			bStarted := TRUE;
			CASE Mode OF
(*------------------ Read parameter ---------------------------------------------------------------*)
				READWRITEPARAMETERMODE_READ	:
					IF NOT fbAdsRead.Busy THEN
						bStarted := FALSE;
						iState := STATE_RUNNING;
					END_IF;
(*------------------ Write parameter ---------------------------------------------------------------*)
				READWRITEPARAMETERMODE_WRITE	:
					IF NOT fbAdsWrite.BUSY THEN
						bStarted := FALSE;
						iState := STATE_RUNNING;
					END_IF;
			END_CASE;
		ELSE
			Done := FALSE;
			ErrorID := MC_ERROR_COMMAND_NOT_ALLOWED;
			Error := TRUE;
		END_IF;

STATE_RUNNING:  (* wait *)
	IF NOT Error THEN
		CASE Mode OF
		(*------------------ Read parameter ---------------------------------------------------------------*)
			READWRITEPARAMETERMODE_READ	:
				IF fbAdsRead.Err THEN
					ValueLreal := 0.0;
					ValueDword := 0;
					ValueBool := FALSE;
					Done := FALSE;
					ErrorID := fbAdsRead.ErrId;
					Error := TRUE;
					fbAdsRead(READ := FALSE);
					iState := STATE_INITIALIZATION;
				ELSE
					Done := TRUE;
					fbAdsRead(READ := FALSE);
			 		iState:=STATE_INITIALIZATION;
				END_IF;
	(*------------------ Write parameter ---------------------------------------------------------------*)
			READWRITEPARAMETERMODE_WRITE	:
				IF fbAdsWrite.Err THEN
					Done := FALSE;
					ErrorID := fbAdsWrite.ErrId;
					Error := TRUE;
					fbAdsWrite(WRITE := FALSE);
					iState := STATE_INITIALIZATION;
				ELSE
					Done := TRUE;
					fbAdsWrite(WRITE := FALSE);
			 		iState:=STATE_INITIALIZATION;
				END_IF;
		END_CASE;
	ELSE
 		iState:=STATE_INITIALIZATION;
	END_IF;

ELSE  (* CASE : Unknown program state *)
	Error := TRUE;
	ErrorID := 16#FFFFFFFF;
	iState:=STATE_INITIALIZATION;
END_CASE;

ADSbusy := fbAdsWrite.BUSY OR fbAdsRead.BUSY;
IF iState=STATE_INITIALIZATION THEN
	(* reset Busy immediately  when sequence ends *)
	Busy := FALSE;
END_IF
END_FUNCTION_BLOCK

(* POU _FBAXIS_REF, ST *)
(*
	AXIS_REF data structure

	The FBAXIS_REF is actually not a function block but a data structure
	It includes the axis I/O variables as well as additional information.
	The reason for not using a STRUCT is that structures cannot hold
	located I/O variables.
	The user is supposed to use the AXIS_REF data type which internally
	redirects the type to this function block definition (alias).
*)
FUNCTION_BLOCK _FBAXIS_REF
VAR_INPUT
	PlcToNc 	AT %Q* 	: 	PLCTONC_AXIS_REF;
END_VAR
VAR_OUTPUT
	NcToPlc 	AT %I* 	:	NCTOPLC_AXIS_REF;
	ADS	 			: 	ST_AdsAddress;
	Status				:	ST_AxisStatus;
END_VAR
{library private}
VAR
	NcCycleCounter: UDINT;
END_VAR
ReadStatus;
END_FUNCTION_BLOCK
ACTION ReadStatus:
(* NC cycle counter will be incremented after NC task updated the NcToPlc data structure *)
NcCycleCounter := SHR(NcToPlc.OpModeDWord, 24);
(* avoid multiple updates during one cycle which would cause additional CPU load *)
IF NcCycleCounter <> Status.NcCycleCounter OR NcCycleCounter=0 THEN
	Status := _F_ReadStatus( NcToPlc := NcToPlc, PlcToNc := PlcToNc );
END_IF
END_ACTION

(* POU _TCMCGLOBAL, ST *)
(*	Global constants and parameters *)
FUNCTION_BLOCK _TCMCGLOBAL
VAR_INPUT
	NCPORT_TCMC 				:	INT 	:= AMSPORT_R0_NC;
	NCPORT_TCMC_COUPLING	:	INT 	:= AMSPORT_R0_NC; (* used with all axis coupling commands - 12.7.2006 KSt *)
	NCNETID_TCMC 				:	T_AmsNetId := '';
	NCPORT_TCMC_CAM 		:	INT 	:= AMSPORT_R0_NC;
	NCNETID_TCMC_CAM		:	T_AmsNetId := '';
END_VAR
VAR_OUTPUT
END_VAR
VAR CONSTANT
	Axis 	: _ST_NCADS_Axis;	(* IDXGRP and IDXOFFS constants of axis parameter/status/functions *)
	Table 	: _ST_NCADS_Table;	(* IDXGRP and IDXOFFS constants of table parameter/status/functions *)

	NCPORT_TCNCCAMMING_TABLEFUNCTION	: 	UINT	:=	500;

	(* timeout *)
	tTargetPosTimeOut			:	TIME	:= T#6s; (* 20050128 KSt - changed from 5 sec to 6 sec to be later than a NC PEH error (5 sec) *)
	tADSTimeOut   				:	TIME	:= T#1s;

	NCTOPLC_FEEDBACK_MAXWAITCYCLES : INT := 10; (* maximum number of PLC cycles to wait for a cyclic feedback in NcToPlc after an ADS command *)
END_VAR
;
END_FUNCTION_BLOCK

(* POU F_AxisCamDataQueued, ST *)
FUNCTION F_AxisCamDataQueued : BOOL
(* 	reference: 	NC -> PLC axis interface (128 bytes)
	check if bit 22 of an axis StateDWord is set:
	New cam data has been queued to a slave axis which is coupled to master via a cam table. 
	The flag comes up when the PLC modifies the camming data.
	Das Flag wird TRUE, wenn neue bzw. veränderte Kurvenscheibendaten von der SPS an 
	eine Slave-Achse gesendet werden.
*)
VAR_INPUT
	StateDWord : DWORD;
END_VAR
VAR
END_VAR
F_AxisCamDataQueued := (StateDWord AND 2#0000_0000_0100_0000_0000_0000_0000_0000) <> 0;
END_FUNCTION

(* POU F_AxisCamScalingPending, ST *)
FUNCTION F_AxisCamScalingPending : BOOL
(* 	reference: 	NC -> PLC axis interface (128 bytes)
	check if bit 23 of an axis StateDWord is set:
	- The flag signals that the scaling and/or offset setting of a cam table has been requested 
	to be performed 	at a certain master position. This request is pending while the function 
	result is TRUE and has been executed after a falling edge of this signal.
	- Das Flag zeigt an das die Skalierung und/oder das Setzen der Offsets einer Kurvenscheibe
	beauftrag wurde aber erst später (ab einer bestimmten Master-Position) durchgeführt wird.
	Mit fallender Flanke des Signals wurde der Auftrag ausgeführt.
*)
VAR_INPUT
	StateDWord : DWORD;
END_VAR
VAR
END_VAR
F_AxisCamScalingPending := (StateDWord AND 2#0000_0000_1000_0000_0000_0000_0000_0000) <> 0;
END_FUNCTION

(* POU F_AxisCamTableQueued, ST *)
FUNCTION F_AxisCamTableQueued : BOOL
(* 	reference: 	NC -> PLC axis interface (128 bytes)
	check if bit 21 of an axis StateDWord is set:
	New cam data has been queued to a slave axis which is coupled to master via a cam table. 
	The flag comes up when the PLC modifies the camming data.
	Das Flag wird TRUE, wenn neue bzw. veränderte Kurvenscheibendaten von der SPS an 
	eine Slave-Achse gesendet werden.
*)
VAR_INPUT
	StateDWord : DWORD;
END_VAR
VAR
END_VAR
F_AxisCamTableQueued := (StateDWord AND 2#0000_0000_0010_0000_0000_0000_0000_0000) <> 0;
END_FUNCTION

(* POU F_AxisExternalLatchValid, ST *)
FUNCTION F_AxisExternalLatchValid : BOOL
(* 	reference: 	NC -> PLC axis interface (128 bytes)
	check if bit 16 of an axis StateDWord is set:
	External latch value or sensing switch has become valid
	Externer Latchwert bzw. Messtaster gültig geworden
*)
VAR_INPUT
	StateDWord : DWORD;
END_VAR
VAR
END_VAR
F_AxisExternalLatchValid := (StateDWord AND 2#0000_0000_0000_0001_0000_0000_0000_0000) <> 0;
END_FUNCTION

(* POU F_AxisGotNewTargetPosition, ST *)
FUNCTION F_AxisGotNewTargetPosition  : BOOL
(* 	reference: 	NC -> PLC axis interface (128 bytes)
	check if bit 17 of an axis StateDWord is set:
	Axis got a new target position or a new velocity
	while the current move command is in execution.
	Die Zielposition oder die Geschwindigkeit der Achse
	wurde geändert, während die Achse eine Bewegung ausführt
*)
VAR_INPUT
	StateDWord : DWORD;
END_VAR
VAR
END_VAR
F_AxisGotNewTargetPosition := (StateDWord AND 2#0000_0000_0000_0010_0000_0000_0000_0000) <> 0;
END_FUNCTION

(* POU F_AxisHasExtSetPointGen, ST *)
FUNCTION F_AxisHasExtSetPointGen : BOOL
(* 	reference: 	NC -> PLC axis interface (128 bytes)
	check if bit 14 of an axis StateDWord is set:
	Axis has an external set point generator (PLC)
	Achse hat einen externen Sollwertgenerator (SPS)
*)
VAR_INPUT
	StateDWord : DWORD;
END_VAR
VAR
END_VAR
F_AxisHasExtSetPointGen := (StateDWord AND 2#0000_0000_0000_0000_0100_0000_0000_0000) <> 0;
END_FUNCTION

(* POU F_AxisInPTPmode, ST *)
FUNCTION F_AxisInPTPmode : BOOL
(* 	reference: 	NC -> PLC axis interface (128 bytes)
	check if bit 25 of an axis StateDWord is set:
	- The flag signals that the axis accepts PTP motion commands. That requires that the axis is 
	not coupled to other axes and not part of a NC-I or FIFO group.
	- Das Flag zeigt an, dass die Achse PTP Bewegungskommandos entgegen nimmt. Das setzt 
	voraus, dass die Achse nicht gekoppelt ist oder in eine NC-I oder FIFO-Gruppe integriert ist.
*)
VAR_INPUT
	StateDWord : DWORD;
END_VAR
VAR
END_VAR
F_AxisInPTPmode := (StateDWord AND 2#0000_0010_0000_0000_0000_0000_0000_0000) <> 0;
END_FUNCTION

(* POU F_AxisIoDataIsInvalid, ST *)
FUNCTION F_AxisIoDataIsInvalid : BOOL
(* 	reference: 	NC -> PLC axis interface (128 bytes)
	check if bit 30 of an axis StateDWord is set:
	Axis I/O data is invalid  (e.g. invalid 'WcState' or 'CdlState' )
	Achse hat keine gültigen I/O-Daten  (e.g. invalid 'WcState' or 'CdlState' )
*)
VAR_INPUT
	StateDWord : DWORD;
END_VAR
VAR
END_VAR
F_AxisIoDataIsInvalid := (StateDWord AND 2#0100_0000_0000_0000_0000_0000_0000_0000) <> 0;
END_FUNCTION

(* POU F_AxisIsCalibrated, ST *)
FUNCTION F_AxisIsCalibrated : BOOL
(* 	reference: 	NC -> PLC axis interface (128 bytes)
	check if bit 1 of an axis StateDWord is set:
	Axis has been referenced ("Axis calibrated")
	Achse ist referenziert ("Achse geeicht")
*)
VAR_INPUT
	StateDWord : DWORD;
END_VAR
VAR
END_VAR
F_AxisIsCalibrated := (StateDWord AND 2#0000_0000_0000_0000_0000_0000_0000_0010) <> 0;
END_FUNCTION

(* POU F_AxisIsMoving, ST *)
FUNCTION F_AxisIsMoving : BOOL
(* 	reference: 	NC -> PLC axis interface (128 bytes)
	check if bit 9 OR 10 of an axis StateDWord is set:
	Axis moving (forward or backwards)
	Achse fährt (vorwärts oder rückwärts)
*)
VAR_INPUT
	StateDWord : DWORD;
END_VAR
VAR
END_VAR
F_AxisIsMoving := (StateDWord AND 2#0000_0000_0000_0000_0000_0110_0000_0000) <> 0;
END_FUNCTION

(* POU F_AxisIsMovingBackwards, ST *)
FUNCTION F_AxisIsMovingBackwards : BOOL
(* 	reference: 	NC -> PLC axis interface (128 bytes)
	check if bit 10 of an axis StateDWord is set:
	Axis moving to logically smaller values
	Achse fährt logisch kleiner
*)
VAR_INPUT
	StateDWord : DWORD;
END_VAR
VAR
END_VAR
F_AxisIsMovingBackwards := (StateDWord AND 2#0000_0000_0000_0000_0000_0100_0000_0000) <> 0;
END_FUNCTION

(* POU F_AxisIsMovingForward, ST *)
FUNCTION F_AxisIsMovingForward : BOOL
(* 	reference: 	NC -> PLC axis interface (128 bytes)
	check if bit 9 of an axis StateDWord is set:
	Axis moving to logically larger values
	Achse fährt logisch größer
*)
VAR_INPUT
	StateDWord : DWORD;
END_VAR
VAR
END_VAR
F_AxisIsMovingForward := (StateDWord AND 2#0000_0000_0000_0000_0000_0010_0000_0000) <> 0;
END_FUNCTION

(* POU F_AxisIsNotMoving, ST *)
FUNCTION F_AxisIsNotMoving : BOOL
(* 	reference: 	NC -> PLC axis interface (128 bytes)
	check if bit 2 of an axis StateDWord is set:
	Axis is logically stationary ("Axis not moving")
	Achse ist im logischen Stillstand ("Achse fährt nicht")
*)
VAR_INPUT
	StateDWord : DWORD;
END_VAR
VAR
END_VAR
F_AxisIsNotMoving := (StateDWord AND 2#0000_0000_0000_0000_0000_0000_0000_0100) <> 0;
END_FUNCTION

(* POU F_AxisJobPending, ST *)
FUNCTION F_AxisJobPending : BOOL
(* 	reference: 	NC -> PLC axis interface (128 bytes)
	check if bit 24 of an axis StateDWord is set:
	- The flag signals that the a new motion job ist pending and will be 
	   executed after the active job is finished (buffer mode)
	- Das Flag zeigt an das die ein neuer Fahrauftrag gepuffert ist,
	   um nach dem aktuellen Auftrag ausgeführt zu werden (buffer mode)
*)
VAR_INPUT
	StateDWord : DWORD;
END_VAR
VAR
END_VAR
F_AxisJobPending := (StateDWord AND 2#0000_0001_0000_0000_0000_0000_0000_0000) <> 0;
END_FUNCTION

(* POU F_AxisReachedConstantVelocity, ST *)
FUNCTION F_AxisReachedConstantVelocity  : BOOL
(* 	reference: 	NC -> PLC axis interface (128 bytes)
	check if bit 12 of an axis StateDWord is set:
	Axis has reached its constant velocity or rotary speed
	Achse hat V-Konst bzw. Drehzahl erreicht
*)
VAR_INPUT
	StateDWord : DWORD;
END_VAR
VAR
END_VAR
F_AxisReachedConstantVelocity := (StateDWord AND 2#0000_0000_0000_0000_0001_0000_0000_0000) <> 0;
END_FUNCTION

(* POU F_GetVersion_TcMC2, ST *)
FUNCTION F_GetVersion_TcMC2 : UINT	(* Gets the library version info *)
VAR_INPUT
	nVersionElement		:	INT;
END_VAR
(*
	Possible nVersionElement parameter:
	1	:	major number
	2	:	minor number
	3	:	revision number
*)

(* Version history:
Date	|	Version/Author |	Remark
----------------------------------------------------------------------------------------------------
11.09.01	|	2.01 JP		|	new version depending on 0.99D
22.11.01	|	2.02 JP		|	new version depending on 0.99F
18.01.02	|	2.03 JP		|	new version depending on 1.0
		|				|	changed names, interfaces, execute behavior
25.01.02	|	2.04 JP		|	no CAMMING, change behavior of MC_Power
07.02.02	|	2.05 JP		|	SetOverride in unit less than 1%
13.02.02	|	2.06 JP		|	New: MC_NewPos and MC_NewPosAndVelo
		|				|	removed MC_MoveAdditive
14.02.02	|	2.07 JP		|	completed: MC_Home, MC_MoveSuperImposed
14.02.02	|	2.08 JP		|	renamed MC_NewPosAndVelo New: MC_SetOverride edge triggered
15.02.02	|	2.09 JP		|	changed: MC_Gear
15.02.02	|	2.10 JP		|	changed: MC_SetOverride
04.04.02	|	2.11 JP		|	changed: done for MC_Home 
		|				|	new: Check TimeOut for MoveAbsolute, MoveRelative, Home
08.03.02	|	2.12 JP		|	changed: new flag inserted 
12.03.02	|	2.13 JP		|	changed: reset of bNotExecute
18.03.02	|	2.14 JP		|	changed: MC_Reset waits for ready
22.03.02	|	2.15 JP		|	changed: MC_Read and Write FBs
26.03.02	|	2.16 JP		|	revised: Read/Write Parameter FBs
27.03.02	|	2.17 JP		|	revised: Read/Write Parameter FBs and Home (calibration cam)
09.04.02	|	2.18 JP		|	changed parameter type of some parameters
17.04.02	|	2.19 JP		|	changed: Read(Bool)Parameter new Input to select read mode
							Boolean parameters can be read with ReadParameter
							changed MC_Power: new input override !!			
23.04.02	|	2.20 JP		|	fixed: MC_Home changed: Behavior of MC_MoveAbsolute/Relative
25.04.02	|	2.21 JP		|	changed: MC_Reset: now not waiting for 'axis is ready'. Check with MC_Power !
26.04.02	|	2.22 JP		|	MC_Home: If Posistion =  DEFAULT_HOME_POSITION --> no set of position
							MC_MoveXX: more detailed error messages
05.07.02	|	2.23 JP		|	new MC_MoveAbsoluteOrRestart: combines MoveAbsolute and NewPos
19.07.02	|	2.24 JP		|	changed: E_STATES ---> E_TCMC_STATES
12.09.02	|	2.25 KST		|	changed: MC_MoveAbsolute and MC_MoveRelative now based on FB_MoveGeneric
							MC_NewPos and MC_NewPosAndVelo based on new FB_NewPosAndVeloGeneric 
							new internal start types in MC_MoveAbsoluteOrRestart (message suppression)
16.09.02	|	2.26 ChristophC|	changed: MC_SetActualPosition due to changes in TcNC.Lib
16.10.02	|	2.27 KST		|	new: MC_ExtSetPointGenEnable and MC_ExtSetPointGenDisable
29.10.02	|	2.28 ChristophC|	MC_Stop and MC_SetActualPosition: Ads port changed from TcMcGlobal.NCPORT_TCMC => AMSPORT_R0_NCSAF
12.11.02	|	2.29 ChristophC|	MC_OverrideFilter function block added
13.12.02	|	2.30 JP		|	several smaller changes: MC_ReadStatus, MC_Stop
22.01.03	|	2.31 KSt		|	new additional function MC_ExtSetPointGenFeed
24.03.03	|	2.32 JP		|	added: MC_GearFloat, corr. MC_ReadBoolParameter (wrong for AxisEnPostionRangeMonitoring)
26.03.03	|	2.33 KSt		|	added: MC_MoveModulo
04.04.03	|	2.34 KSt		|	changed: MC_MoveAbsoluteOrRestart, Done will be reset at once after Execute=FALSE
12.05.03	|	2.35 JP		|	changed: MC_MoveVelocity, MC_Home (error handling), MC_ReadStatus
14.05.03	|	2.36 KSt		|	changed: MC_Home, MC_MoveAbsoluteOrRestart
15.05.03	|	2.36.1 KSt	|	changed: MC_Home
28.05.03	|	2.37 KSt		|	changed: MC_MoveVelocity, abort during acceleration phase	
							changed: MC_MoveAbsoluteOrRestart, reset internal error on restart
27.06.03	|	2.38 JP		|	changed: MC_Stop: Execute behavior
22.07.03	|	2.38.1 KSt	|	added: new error codes
12.08.03	|	2.39 KSt		|	changed: FB_ReadWriteParameter, size of bool parameters
15.08.03	|	2.40 KSt		|	added: new block MC_ChangeDynParam
19.08.03	|	2.41 JP		|	changed: MC_ReadParameter: Done falls with Execute
01.10.03	|	2.42 KSt		|	changed: MC_MoveAbsoluteOrRestart, Execute directly after done issue fixed
09.10.03	|	2.43 KSt		|	new function block MC_SetReferenceFlag
04.12.03	|	2.44 KSt		|	ReadBoolParameter(AxisEnTargetPositionMonitoring) corrected
12.01.04	|	2.45 KSt		|	MC_MoveSuperimposed revised
						|	R_Trigger(execute) moved outside CASE in all move function blocks
19.01.04	|	2.45.1 KSt	|	Busy Signal in MC_MoveSuperimposed
30.04.04	|	2.46.0 KSt	|	New function blocks MC_TouchProbe, MC_AbortTrigger, internal block MC_OrientedStop
						|	MC_ReadParameter revised
06.05.04	|	2.46.1 KSt	|	Correction in MC_OrientedStop
21.05.04	|	2.47.0 KSt	|	MC_GearInDyn added - master slave coupling with dynamic gear ratio
06.08.04	|	2.47.1 KSt	|	MC_OrientedStop moved from internal to additional folder
						|	MC_MoveAbsoluteOrRestart additional internal error code NC_ERROR_STARTINTERNAL_NOTREADY evaluated
23.08.04	|	2.47.2 KSt	|	new local flag EmergencyStop in MC_Stop signals type of internal ADS stop command
10.01.05	|	2.47.3 KSt	|	new function block MC_MoveSuperImposedExt
28.01.05	|	2.47.4 KSt	|	TcMcGlobal.tTargetPosTimeOut changed from 5 sec to 6 sec to be later than a NC PEH error (5 sec)
15.02.05	|	2.48.0 KSt	|	new function block MC_GearOutExt 
28.02.05	|	2.49.0 JP		|	Execute and Done behavior corrected for MC_ReadActualPos and MC_SetActualPos
10.03.05	|	2.50.0 KSt	|	all function blocks use a global AMS net-ID TcMcGlobal.NCNETID_TCMC which may be modified by the user
17.03.05	|	2.51.0 KSt	|	new function block MC_PowerStepper
						|	MC_MoveAbsoluteOrRestart restart while starting (adswrite.Busy) changed
24.05.05	|	2.52.0 KSt	|	acceleration added to block MC_GearOutExt 
05.07.05	|	2.53.0 KSt	|	new local flag ADSbusy in all function blocks
05.07.05	|	2.54.0 KSt	|	new function block MC_GearInDynCCV
06.07.05	|	2.55.0 KSt	|	Busy timing improved in all function blocks (turns immediately to FALSE with Done or Error or Aborted)
25.07.05	|	2.55.1 KSt	|	Change for status output behavior 
26.07.05	|	2.55.2 KSt	|	MC_GearOutExt extended through mode 'oriented stop'
03.08.05	|	2.55.3 KSt	|	Commands MC_MoveAbsoluteOrRestart, MC_NewPos and MC_NewPosAndVelo now directed to port AMSPORT_R0_NCSAF
						|	Summary of other commands to SAF: MC_Stop, MC_OrientedStop, MC_TouchProbe, MC_AbortTrigger, MC_SetReferenceFlag, MC_PowerStepper
14.09.05	|	2.56.0 KSt	|	new function block MC_ParameterizedStop
26.09.05	|	2.56.1 KSt	|	Jerk parameter added to MC_ChangeDynParam. Block moved into the internal folder.
07.11.05	|	2.56.2 KSt	|	internal block FB_ReadCharacteristicValues changed to ADSRDWRT
19.12.05	|	2.56.3 KSt	|	new block MC_SetActualPositionOnTheFly
05.01.06	|	2.56.4 KSt	|	new blocks MC_ReadParameterSet and MC_ReadAxisComponents
21.02.06	|	2.57.0 KSt	|	NC status feedback monitoring changed in MC_GearIn and MC_GearInFloat
29.03.06	|	2.57.1 KSt	|	new order of the blocks in the library tree
11.04.06	|	2.57.2 HKP	|	Command MC_ChangeDynParam now directed to port AMSPORT_R0_NCSAF
10.05.06	|	2.57.3 KSt	|	new function block MC_Jog
17.05.06	|	2.57.4 KSt	|	MC_Jog: MC_JOGMODE_INCHING_MODULO temporarily deactivated
05.07.06	|	2.57.5 KSt	|	NC status feedback monitoring changed in MC_GearInDyn and MC_GearInDynCCV
=======	|===============	|==========================================================================
12.07.06	|	2.57.6 KSt	|	new AMS port NCPORT_TCMC_COUPLING for all coupling commands
11.08.06	|	2.57.7 KSt	|	reset Done when Execute is FALSE in FB_NewPosAndVeloGeneric
						|	MC_Jog released
22.08.06	|	2.57.8 KSt	|	new function block MC_AbortSuperposition
07.11.06	|	2.57.9 HKP	|	changes in function block MC_PowerStepper
06.02.07	|	2.57.10 KSt	|	initialization problem with modulo positions fixed in MC_TouchProbe.
						|	recorded position at PlcEvent now modulo when requested.
14.03.07	|	2.57.11 KSt	|	MC_Jog: Handling of CommandAborted corrected
24.04.07	|	2.57.12 KSt	|	additional parameters in MC_AxisPara, MC_ReadParameters, MC_WriteParameters
31.05.07	|	2.57.13 KSt	|	FPU exception with LREAL_TO_BOOL and DWORD_TO_BOOL fixed in FB_ReadWriteParameter 
12.06.07	|	2.57.14 KSt	|	FB_NewPosAndVeloGeneric and MC_MoveSuperImposed(Ext): IF condition changed from "NOT AxisIsMoving" to "NOT AxisHasJob"
=======	|===============	|==========================================================================
12.06.07	|	2.57.14 KSt	|	TcMC2 development started - following 2.xx.xx changes have been added in parallel
02.11.07	|	2.57.15 KSt	|	data structure ST_TableCharacValues extended
18.12.07	|	2.57.16 KSt	|	MC_Jog is now internally using MC_MoveRelative instead of MC_MoveAbsolute to work with backlash compensation
20.05.08	|	2.57.18 KSt	|	AxisModuloPositionFlag added to MC_ReadBoolParameter
17.06.08	|	2.57.20 KSt	|	MC_GearInMultiMaster added
24.07.08	|	2.57.22 KSt	|	MC_Power supports now a minimum Enable-Off/On toggle time of 50ms to reenable the Status output
28.10.08	|	2.57.23 KSt	|	new function block MC_SetEncoderScalingFactor
=======	|===============	|==========================================================================
16.03.07	|	3.00.00 KSt	|	new version depending on PLCopen V1.1 (beta)
25.08.08   |	3.00.01 KSt	|	released as TcMC2 
17.09.08   |	3.00.02 KSt	|	last result added in MC_Reset
26.11.08   |	3.00.03 KSt	|	change in MC_Stop and MoveGeneric for delayed error handling
01.12.08   |	3.00.04 KSt	|	MC_Stop - Done is set immediately at standstill
18.12.08   |	3.00.05 KSt	|	MC_Power - uses now ControlLoopClosed instead of AxisIsReady
13.01.09   |	3.00.06 KSt	|	independent characteristic data for camming and flying saw
16.01.09   |	3.00.07 KSt	|	all move commands: changed handling of CmdNo=0 and CmdNo+2 leads to better results (CommandAborted)
23.01.09   |	3.00.08 KSt	|	MC_MoveSuperimposed is now passed to port AMSPORT_R0_NCSAF (501)
28.01.09   |	3.00.09 KSt	|	Homing mode MC_Direct added - Mode option for MC_SetPosition added
29.01.09   |	3.00.10 KSt	|	Warning output added to MC_MoveSuperimposed
05.02.09   |	3.00.11 KSt	|	axis state is now DISABLED if control loop is not closed (was STANDSTILL for virtual axes - _F_AxisState)
05.02.09   |	3.00.11 KSt	|	all move commands: CmdNo=0 is ignored as invalid - change of the coupled state leads to CommandAborted
06.02.09   |	3.00.11 KSt	|	errors on missing cyclic NC command feedback are delayed for a few cycles to avoid problems with multiple function block calls during one PLC cycle
19.02.09   |	3.00.12 KSt	|	MC_GearInDyn and MC_GearInMultimaster - no reset of gear ratio after Enable is reset to FALSE
24.02.09   |	3.01.00 KSt	|	Motion commands on slaves (must be enabled in the axis parameters before)
12.03.09   |	3.01.01 KSt	|	MC_Jog - Active output added - reset outputs when Execute is false 
09.04.09   |	3.01.02 KSt	|	MC_SetPosition and MC_SetEncoderScalingFactor - explicit encoder / control loop index 0..n can be selected
15.04.09   |	3.01.03 KSt	|	MC_Stop - outputs (except Busy) are reset after Execute=FALSE - can be retriggered during release phase
17.04.09   |	3.01.04 KSt	|	MC_Home - static homing with DEFAULT_HOME_POSITION implemented - Option.ClearPositionLag available 
11.05.09   |	3.01.05 KSt	|	MC_Stop - incorrect error message 4B63 removed;  
30.06.09   |	3.01.06 KSt	|	MC_MoveSuperimposed - new types ACCREDUCTION - new AbortOptions
28.07.09   |	3.01.07 KSt	|	MC_ExtSetPointGenFeed feeds additional counter information to the NC
13.08.09   |	3.01.08 KSt	|	MC_MoveSuperimposed - new AbortOptions - Done behavior adapted
01.09.09   |	3.01.09 KSt	|	MC_SetPosition - new option 'set absolute measuring'
30.09.09   |	3.01.10 KSt	|	MC_MoveSuperimposed - fix for new AbortOptions - HasJob flag not required before starting the command
06.10.09   |	3.01.11 KSt	|	MC_Stop - wait extra cycles before axis release error 
06.10.09   |	3.01.12 KSt	|	MC_MoveSuperimposed - fix for new AbortOptions - HasJob or IsMoving check at beginning and end of compensation 
07.10.09   |	3.01.13 KSt	|	MC_MoveSuperimposed - initial motion check removed for new AbortOptions
28.10.09   |	3.01.14 KSt	|	MC_ExtSetPointGenEnable/Disable - port changed from SVB to SAF
06.11.09   |	3.01.15 KSt	|	MC_SetPosition - new option 'set absolute measuring' removed
09.11.09   |	3.01.16 KSt	|	MC_Stop on slave axes was not rejected with error - fixed
18.11.09   |	3.01.17 KSt	|	MC_Jog - usage with protected (coupled) axes refused
26.11.09   |	3.01.18 KSt	|	Axis status data: UpdateCycleTime calculation fixed
08.12.09   |	3.01.19 KSt	|	_FB_MoveGeneric - mapping check to avoid early Error and CommandAborted signals
25.02.10   |	3.01.20 KSt	|	MC_MoveSuperimposed - additional outputs ActualAcceleration and ActualDeceleration
11.03.10   |	3.01.21 KSt	|	MC_Power - no Enable timeout error for coupled axes
*)
CASE nVersionElement OF
1:	(* major number *)
	F_GetVersion_TcMC2 := 3;
2:	(* minor number *)
	F_GetVersion_TcMC2 := 1;
3:	(* revision number *)
	F_GetVersion_TcMC2 := 21;
ELSE
	F_GetVersion_TcMC2 := 16#FFFF;
END_CASE
END_FUNCTION

(* POU MC_AbortSuperposition, ST *)
FUNCTION_BLOCK MC_AbortSuperposition
VAR_INPUT
	Execute		:	BOOL;	(* Starts touch probe recording *)
END_VAR
VAR_OUTPUT
	Done		:	BOOL;	(* move completed *)
	Busy		: 	BOOL;	(* function block is currently Busy *)
	Error		:	BOOL;	(* Signals that error has occured within Function Block *)
	ErrorID		:	UDINT;	(* Error identification *)
END_VAR
VAR_IN_OUT
	Axis			:	AXIS_REF; (* Identifies the axis of which the position should be recorded at a defined event at the trigger input *)
END_VAR
VAR
	LastExecutionResult: 	_ST_FunctionBlockResults;
	ADSbusy	: 	BOOL;
	fbOnTrigger	: 	R_TRIG;
	fbADSwrite	: 	ADSWRITE;
	iState		:	_E_TcMC_STATES := STATE_INITIALIZATION;
END_VAR
fbOnTrigger(CLK:= Execute);

CASE iState OF
STATE_INITIALIZATION: (* initial iState *)
	Busy := FALSE;
	IF NOT Execute THEN
		Done := FALSE;
		Error := FALSE;
		ErrorID := 0;
	END_IF
	IF fbOnTrigger.Q THEN
		Busy := TRUE;
		(* initialization *)
		Done := FALSE;
		Error := FALSE;
		ErrorID := 0;
		LastExecutionResult.Done := FALSE;
		LastExecutionResult.CommandAborted := FALSE;
		LastExecutionResult.Error := FALSE;
		LastExecutionResult.ErrorID := 0;
		fbADSwrite(WRITE:=FALSE);
		fbADSwrite(	NETID:= TcMcGlobal.NCNETID_TCMC,
					PORT:=TcMcGlobal.NCPORT_TCMC ,
					IDXGRP:= TcMcGlobal.Axis.Functions.IDXGRP + Axis.NcToPlc.AxisId,
					IDXOFFS:= TcMcGlobal.Axis.Functions.IDXOFFS.STOPSCOM,	(* abort superposition *)
					LEN:=0,
					SRCADDR:=0,
					WRITE:=TRUE ,
					TMOUT:= TcMcGlobal.tADSTimeOut);
		iState := STATE_ORDER;
	END_IF

STATE_ORDER:  (* wait until command is accepted *)
	fbADSwrite(WRITE:= TRUE);
	IF NOT fbADSwrite.BUSY THEN
		Error := fbADSwrite.ERR;
		ErrorID := fbADSwrite.ERRID;
		IF NOT Error THEN
			IF NOT F_AxisIsCompensating(Axis.NcToPlc.StateDWord) THEN
				Done := TRUE;
				Busy := FALSE;
				iState := STATE_INITIALIZATION;
			ELSE
				iState := STATE_RUNNING;
			END_IF
		ELSE
			Busy := FALSE;
			iState := STATE_INITIALIZATION;
		END_IF
		LastExecutionResult.Done := Done;
		LastExecutionResult.Error := Error;
		LastExecutionResult.ErrorID := ErrorID;
	END_IF

STATE_RUNNING:
	IF NOT F_AxisIsCompensating(Axis.NcToPlc.StateDWord) THEN
		Done := TRUE;
		Busy := FALSE;
		LastExecutionResult.Done := Done;
		LastExecutionResult.Error := Error;
		LastExecutionResult.ErrorID := ErrorID;
		iState := STATE_INITIALIZATION;
	END_IF
END_CASE

ADSbusy := fbAdsWrite.BUSY;
END_FUNCTION_BLOCK

(* POU MC_AbortTrigger, ST *)
FUNCTION_BLOCK MC_AbortTrigger
(*	The function block is used to abort function blocks which are connected to
	trigger events (e.g. MC_TouchProbe) 
*)
VAR_IN_OUT
	Axis			:	AXIS_REF; 		(* B *)	(* Identifies the axis of which the position should be recorded at a defined event at the trigger input *)
	TriggerInput	: 	TRIGGER_REF; 	(* E *)	(* Reference to the trigger signal source. *)
END_VAR
VAR_INPUT
	Execute		:	BOOL;	(* B *)	(* Starts aborting  touch probe sequence *)
END_VAR
VAR_OUTPUT
	Done		:	BOOL;	(* B *)	(* function completed *)
	Busy		: 	BOOL;	(* E *)	(* function block is currently Busy *)
	Error		:	BOOL;	(* B *)	(* Signals that error has occurred within Function Block *)
	ErrorID		:	UDINT;	(* E *)	(* Error identification *)
END_VAR
VAR
	ADSbusy	: 	BOOL;
	fbADSwrite	: 	ADSWRITE;
END_VAR
{library private}
VAR CONSTANT
	OLDADSINTERFACE : BOOL := TRUE; (* temporary flag to test old and new NC ADS touch probe interface *)
END_VAR
VAR
	LatchID		: 	UDINT;
	fbOnTrigger	: 	R_TRIG;
END_VAR
IF NOT Execute THEN
	Done := FALSE;
	Error := FALSE;			(* reset at falling edge of Execute *)
	ErrorID := 0;
END_IF

fbOnTrigger(CLK:= Execute);
IF fbOnTrigger.Q OR fbADSwrite.BUSY THEN
	Busy := TRUE;
	IF fbOnTrigger.Q THEN
		(* initialization *)
		Done := FALSE;
		Error := FALSE;
		ErrorID := 0;
		fbADSwrite(WRITE:=FALSE);
		IF TriggerInput.EncoderID > 255 THEN
			Error := TRUE;
			ErrorID := MC_ERROR_INVALID_TOUCH_PROBE;
		END_IF
	END_IF

	IF NOT Error THEN
		CASE TriggerInput.TouchProbe OF
			TouchProbe1,
			TouchProbe2,
			TouchProbe3,
			TouchProbe4:
			LatchID := TriggerInput.TouchProbe;
			fbADSwrite(	NETID:= TcMcGlobal.NCNETID_TCMC,
						PORT:=AMSPORT_R0_NCSAF ,
						IDXGRP:=16#5200+TriggerInput.EncoderID ,
						IDXOFFS:=16#205,	(* deactivate touch probe *)
						LEN:=SEL(OLDADSINTERFACE, SIZEOF(LatchID), 0) ,
						SRCADDR:=ADR(LatchID),
						WRITE:=TRUE ,
						TMOUT:=TcMcGlobal.tADSTimeOut);
			IF NOT fbADSwrite.BUSY THEN
				Error := fbADSwrite.ERR;
				ErrorID := fbADSwrite.ERRID;
				TriggerInput.ProbeState := SEL(Error, TouchProbeAborted, TriggerInput.ProbeState );
				Done := NOT Error;
			END_IF

			PlcEvent:
				(* no action necessary here *);
				TriggerInput.ProbeState := TouchProbeAborted;
				Done := TRUE;

			ELSE (* case *)
				Error := TRUE;
				ErrorID := MC_ERROR_INVALID_TOUCH_PROBE;
		END_CASE
	END_IF
ELSE
	Busy := FALSE;
END_IF

ADSbusy := fbAdsWrite.BUSY;
(* reset Busy immediately  when sequence ends *)
Busy := fbOnTrigger.Q OR fbADSwrite.BUSY;
END_FUNCTION_BLOCK

(* POU MC_ExtSetPointGenDisable, FBD *)
FUNCTION_BLOCK MC_ExtSetPointGenDisable
VAR_IN_OUT
	Axis	:	AXIS_REF;
END_VAR
VAR_INPUT
	Execute : BOOL;
END_VAR
VAR_OUTPUT
	Done : BOOL;
	Busy: BOOL;
	Error: BOOL;
	ErrorID: UDINT;
	Enabled: BOOL;
END_VAR
VAR
	ADSbusy: BOOL;
	Disable: ADSWRITE;
	RunOnce: BOOL;
END_VAR
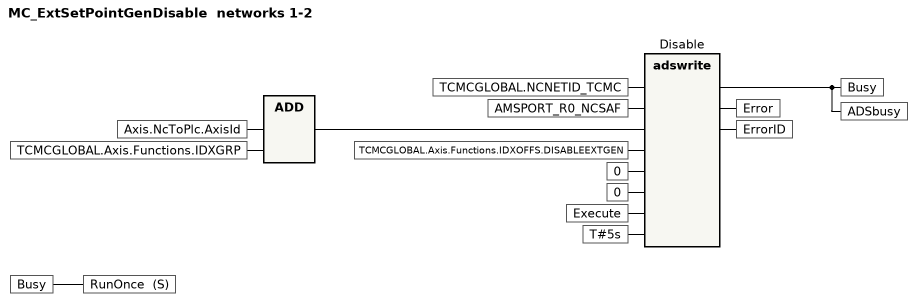
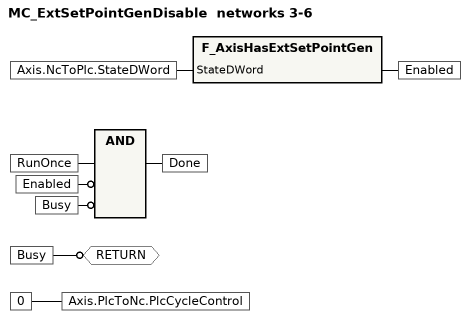
_FBD_ (* Function Block Diagram *)
NETWORK 1 (* ( * 2009-10-28 KSt - port changed from SVB to SAF * ) *)
	Disable:adswrite(TCMCGLOBAL.NCNETID_TCMC, AMSPORT_R0_NCSAF, ADD(Axis.NcToPlc.AxisId, TCMCGLOBAL.Axis.Functions.IDXGRP), TCMCGLOBAL.Axis.Functions.IDXOFFS.DISABLEEXTGEN, 0, 0, Execute, T#5s, out 2 => Error, out 3 => ErrorID) => Busy, ADSbusy
NETWORK 2
	Busy => S RunOnce
NETWORK 3
	F_AxisHasExtSetPointGen(StateDWord: Axis.NcToPlc.StateDWord) => Enabled
NETWORK 4
	AND(RunOnce, NOT Enabled, NOT Busy) => Done
NETWORK 5
	NOT Busy => <RETURN>
NETWORK 6
	0 => Axis.PlcToNc.PlcCycleControl
_END_FBD_
END_FUNCTION_BLOCK

(* POU MC_ExtSetPointGenEnable, FBD *)
FUNCTION_BLOCK MC_ExtSetPointGenEnable
VAR_IN_OUT
	Axis	:	AXIS_REF;
END_VAR
VAR_INPUT
	Execute : BOOL;
	Position : LREAL;
	PositionType : E_PositionType;
END_VAR
VAR_OUTPUT
	Done : BOOL;
	Busy: BOOL;
	Error: BOOL;
	ErrorID: UDINT;
	Enabled: BOOL;
END_VAR
VAR
	ADSbusy: BOOL;
	Enable: ADSWRITE;
	sExtSetPointGen : _ST_TcNC_SetPos;
END_VAR
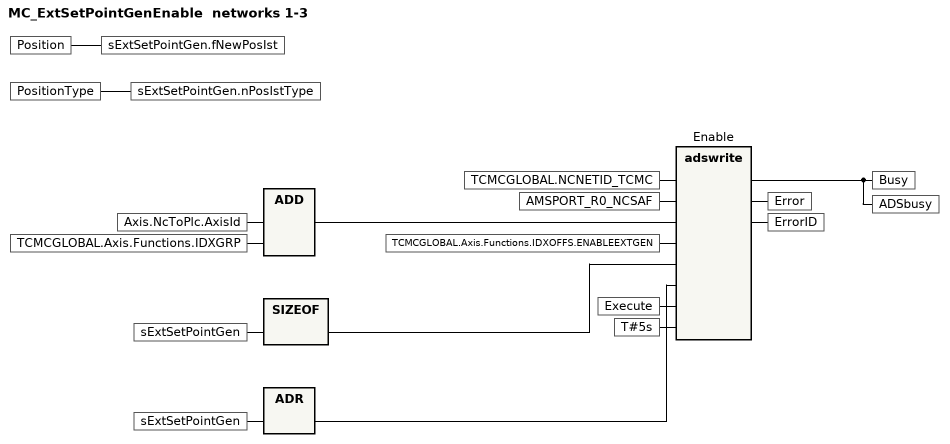
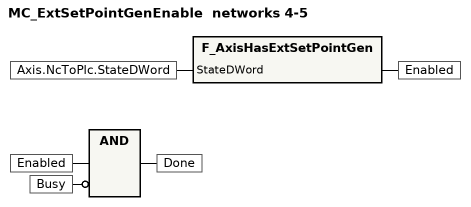
_FBD_ (* Function Block Diagram *)
NETWORK 1
	Position => sExtSetPointGen.fNewPosIst
NETWORK 2
	PositionType => sExtSetPointGen.nPosIstType
NETWORK 3 (* ( * 2009-10-28 KSt - port changed from SVB to SAF * ) *)
	Enable:adswrite(TCMCGLOBAL.NCNETID_TCMC, AMSPORT_R0_NCSAF, ADD(Axis.NcToPlc.AxisId, TCMCGLOBAL.Axis.Functions.IDXGRP), TCMCGLOBAL.Axis.Functions.IDXOFFS.ENABLEEXTGEN, SIZEOF(sExtSetPointGen), ADR(sExtSetPointGen), Execute, T#5s, out 2 => Error, out 3 => ErrorID) => Busy, ADSbusy
NETWORK 4
	F_AxisHasExtSetPointGen(StateDWord: Axis.NcToPlc.StateDWord) => Enabled
NETWORK 5
	AND(Enabled, NOT Busy) => Done
_END_FBD_
(* the same logic as Structured Text *)
(* Network 1 *)
sExtSetPointGen.fNewPosIst := Position;
(* Network 2 *)
sExtSetPointGen.nPosIstType := PositionType;
(* Network 3: see the listing above *)
(* Network 4 *)
Enabled := F_AxisHasExtSetPointGen(StateDWord := Axis.NcToPlc.StateDWord);
(* Network 5 *)
Done := Enabled AND NOT Busy;
END_FUNCTION_BLOCK

(* POU MC_ExtSetPointGenFeed, ST *)
FUNCTION MC_ExtSetPointGenFeed : BOOL
VAR_IN_OUT
	Axis	:	AXIS_REF;
END_VAR
VAR_INPUT
	Position		: LREAL;
	Velocity		: LREAL;
	Acceleration	: LREAL;
	Direction 	: DINT;
END_VAR
VAR
	GetTaskIndex : GETCURTASKINDEX;
END_VAR
Axis.PlcToNc.ExtSetPos := Position;
Axis.PlcToNc.ExtSetVelo := Velocity;
Axis.PlcToNc.ExtSetAcc := Acceleration;
Axis.PlcToNc.ExtSetDirection := Direction;

GetTaskIndex();
Axis.PlcToNc.PlcCycleControl.0 := 1; (* activate PLC cycle information to NC *)
Axis.PlcToNc.PlcCycleControl.1 := SystemTaskInfoArr[ GetTaskIndex.index ].cycleTimeExceeded;
Axis.PlcToNc.PlcCycleCount := Axis.PlcToNc.PlcCycleCount + 1;
END_FUNCTION

(* POU MC_GearIn, ST *)
FUNCTION_BLOCK MC_GearIn
(*	This Function Block commands a ratio between the velocity of the slave and master axis. *)
VAR_IN_OUT
	Master			:	AXIS_REF;	(* B *)
	Slave			:	AXIS_REF;	(* B *)
END_VAR
VAR_INPUT
	Execute			:	BOOL;	(* B *)
	RatioNumerator	:	LREAL	(* B *)	:= 1; (* changed from INT (PLCopen) to LREAL *)
	RatioDenominator	:	UINT	(* B *)	:= 1;
	Acceleration		:	LREAL;	(* E *)
	Deceleration		:	LREAL;	(* E *)
	Jerk				:	LREAL;	(* E *)
	BufferMode		:	MC_BufferMode;	(* E *)
	Options			: 	ST_GearInOptions;	(* V *)	(* optional parameters *)
END_VAR
VAR_OUTPUT
	InGear			:	BOOL;	(* B *)
	Busy			: 	BOOL;	(* E *)
	Active			: 	BOOL;	(* E *)
	CommandAborted	:	BOOL;	(* E *)
	Error			:	BOOL;	(* B *)
	ErrorID			:	UDINT;	(* E *)
END_VAR
VAR
	LastExecutionResult	: 	_ST_FunctionBlockResults;
	ADSbusy: BOOL;
	iState				:	_E_TcMC_STATES := STATE_INITIALIZATION;
	fbAdsWrite			:	ADSWRITE;
	sCouple				:	_ST_TcNC_CoupleSlave;
	fbOptGearInDyn		: 	MC_GearInDyn;
END_VAR
{library private}
VAR
	fbOnTrigger			:	R_TRIG;
	TimerStateFeedback	: 	TON;
END_VAR
fbOnTrigger(CLK:= Execute);

CASE iState OF
STATE_INITIALIZATION:	(* *)
	Busy := FALSE;
	IF NOT Execute THEN
		InGear := FALSE;
		CommandAborted := FALSE;
		Error := FALSE;			(* reset at falling edge of Execute *)
		ErrorID := 0;
	END_IF
	IF fbOnTrigger.Q THEN
		Busy := TRUE;
		(* initialize output values *)
		InGear 			:= FALSE;
		CommandAborted	:= FALSE;
		ErrorID := 0;
		Error := FALSE;
		LastExecutionResult.Done := FALSE;
		LastExecutionResult.CommandAborted := FALSE;
		LastExecutionResult.Error := FALSE;
		LastExecutionResult.ErrorID := 0;
		fbOptGearInDyn.Enable := FALSE;
		TimerStateFeedback(IN:=FALSE);

		IF RatioDenominator = 0 THEN
			Error := TRUE;
			ErrorID := MC_ERROR_PARAMETER_NOT_CORRECT;
		ELSIF BufferMode <> 0 THEN
			Error := TRUE;
			ErrorID := MC_ERROR_BUFFERMODE_NOT_SUPPORTED;
		ELSE
			CASE Options.SlaveType OF
				0, TCNC_SLAVETYPE_LINEAR :
					(* linear gear ratio coupling *)
					sCouple.nSlaveType 		:= TCNC_SLAVETYPE_LINEAR; (* linear coupling *)
					sCouple.nMasterAxisId		:= Master.NcToPlc.AxisId;
					sCouple.nMasterSubIdx	:= 0;
					sCouple.nSlaveSubIdx		:= 0;
					sCouple.fCoupleParam1	:= RatioNumerator / RatioDenominator;
					sCouple.fCoupleParam2	:= 0;(* unused *)
					sCouple.fCoupleParam3	:= 0;(* unused *)
					sCouple.fCoupleParam4	:= 0;(* unused *)
		
					fbAdsWrite(	NETID:= TcMcGlobal.NCNETID_TCMC,
							PORT:= TcMcGlobal.NCPORT_TCMC_COUPLING,
							IDXGRP:=TcMcGlobal.Axis.Functions.IDXGRP+Slave.NcToPlc.AxisId,
							IDXOFFS:= TcMcGlobal.Axis.Functions.IDXOFFS.CPL,
							LEN:= SIZEOF(sCouple),
							SRCADDR:= ADR(sCouple),
							WRITE:= TRUE,
							TMOUT:= TcMcGlobal.tADSTimeOut);
					iState := STATE_ORDER;

				TCNC_SLAVETYPE_LINEAR_CYCLICCHANGES_RAMP,
				TCNC_SLAVETYPE_CONST_SURFACEVELO_RAMP :
					fbOptGearInDyn.Enable := TRUE;
					ActGearInDyn;
					iState := STATE_ORDER;
			ELSE
				Error := TRUE;	(* Optional mode not supported with this function block *)
				ErrorID := MC_ERROR_PARAMETER_NOT_CORRECT;
			END_CASE
		END_IF;
	END_IF;

STATE_ORDER:
	CASE Options.SlaveType OF
		0, TCNC_SLAVETYPE_LINEAR :
			fbAdsWrite();
			IF NOT fbAdsWrite.Busy THEN
				IF fbAdsWrite.Err THEN
					ErrorID := fbAdsWrite.ErrId;
					Error := TRUE;
					iState := STATE_INITIALIZATION;
				ELSE
					iState := STATE_RUNNING;
				END_IF
				fbAdsWrite(WRITE := FALSE);
			END_IF;

		(* optional modes to couple with dynamically changable gear ratio (just couple) *)
		TCNC_SLAVETYPE_LINEAR_CYCLICCHANGES_RAMP,
		TCNC_SLAVETYPE_CONST_SURFACEVELO_RAMP :
			ActGearInDyn;
			IF fbOptGearInDyn.InGear THEN
				InGear := TRUE;
				fbOptGearInDyn.Enable := FALSE;
				ActGearInDyn;
				iState := STATE_INITIALIZATION;
			ELSIF NOT fbOptGearInDyn.Busy THEN
				CommandAborted := fbOptGearInDyn.CommandAborted;
				Error := fbOptGearInDyn.Error;
				ErrorID := fbOptGearInDyn.ErrorID;
				fbOptGearInDyn.Enable := FALSE;
				iState := STATE_INITIALIZATION;
			END_IF
	ELSE
		Error := TRUE;	(* Optional mode not supported with this function block *)
		ErrorID := MC_ERROR_PARAMETER_NOT_CORRECT;
		iState := STATE_INITIALIZATION;
	END_CASE

STATE_RUNNING:  (* Return *)
	TimerStateFeedback(IN:=TRUE, PT:=t#50ms); (* 21.2.2006 KSt *)
	IF  (Slave.NcToPlc.CoupleState = 2) OR (Slave.NcToPlc.CoupleState = 3) THEN
		(* axis successfully coupled *)
		InGear := TRUE;
		iState := STATE_INITIALIZATION;
	ELSIF TimerStateFeedback.Q THEN
		(* 	nCoupleState does not respond 'coupled' - the reason may be
			a MC_GearOut command which aborted the GearIn command *)
		CommandAborted := TRUE;
		iState := STATE_INITIALIZATION;
	END_IF;

ELSE  (* CASE : Unknown program state *)
	Error := TRUE;
	ErrorID := 16#FFFFFFFF;
	iState:= STATE_INITIALIZATION;
END_CASE

ADSbusy := fbAdsWrite.BUSY;
IF iState=STATE_INITIALIZATION THEN
	(* reset Busy immediately  when sequence ends *)
	IF Busy THEN
		LastExecutionResult.Done := InGear;
		LastExecutionResult.CommandAborted := CommandAborted;
		LastExecutionResult.Error := Error;
		LastExecutionResult.ErrorID := ErrorID;
	END_IF
	Busy := FALSE;
END_IF

Active := Busy;
END_FUNCTION_BLOCK
ACTION ActGearInDyn:
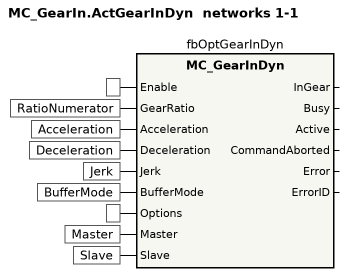
_FBD_ (* Function Block Diagram *)
NETWORK 1
	fbOptGearInDyn:MC_GearInDyn(Enable: , GearRatio: RatioNumerator, Acceleration: Acceleration, Deceleration: Deceleration, Jerk: Jerk, BufferMode: BufferMode, Options: , Master: Master, Slave: Slave)
_END_FBD_
END_ACTION
ACTION WriteGearRatio:
	(* action can be called from external in case of coupling modes with dynamically changable gear ratio *)
	IF RatioDenominator = 0 THEN
		Slave.PlcToNc.AxisModeLReal := RatioNumerator;
	ELSE
		Slave.PlcToNc.AxisModeLReal := RatioNumerator / RatioDenominator;
	END_IF
END_ACTION

(* POU MC_GearInDyn, ST *)
FUNCTION_BLOCK MC_GearInDyn
(*	MC_GearInDyn couples a slave axis to a master axis
 *	using a floating point gear ratio. The gear ratio can be 
 *	dynamically modified every PLC cycle as long as the 
 *	Execute input is TRUE.
 *	The acceleration input specifies the maximum slave
 *	acceleration in case of high gear ratio changes.
 *)
VAR_IN_OUT
	Master			:	AXIS_REF;
	Slave			:	AXIS_REF;
END_VAR
VAR_INPUT
	Enable			:	BOOL;
	GearRatio		:	LREAL := 1.0;
	Acceleration		:	LREAL;
	Deceleration		:	LREAL;	(* not used *)
	Jerk				:	LREAL;	(* not used *)
	BufferMode		:	MC_BufferMode;	(* E *)
	Options			: 	ST_GearInDynOptions;	(* V *)	(* optional parameters *)
END_VAR
VAR_OUTPUT
	InGear				:	BOOL;
	Busy				: 	BOOL;
	Active				: 	BOOL;
	CommandAborted		:	BOOL;
	Error				:	BOOL;
	ErrorID				:	UDINT;
END_VAR
VAR
	LastExecutionResult: 	_ST_FunctionBlockResults;
	ADSbusy: BOOL;
	iState			:	_E_TcMC_STATES := STATE_INITIALIZATION;
	iSubState		: 	INT;
	fbAdsWrite		:	ADSWRITE;
	fbAdsRead		:	ADSREAD;
	sCouple			:	_ST_TcNC_CoupleSlave;
	v_max			: 	LREAL;
	pa_limit			: 	LREAL;
	WasInGear: BOOL;
END_VAR
{library private}
VAR
	iAcceleration		: 	LREAL;
	TimerStateFeedback: TON;
END_VAR
CASE iState OF
	STATE_INITIALIZATION:	(* *)
		Busy := FALSE;
		Active := FALSE;
		IF Enable THEN
			Busy := TRUE;
			Active := TRUE;
			fbAdsRead(READ:=FALSE);
			fbAdsWrite(WRITE:=FALSE);
			(* initialize output values *)
			iAcceleration := Acceleration;
			ErrorID := 0;
			Error := FALSE;
			LastExecutionResult.Done := FALSE;
			LastExecutionResult.CommandAborted := FALSE;
			LastExecutionResult.Error := FALSE;
			LastExecutionResult.ErrorID := 0;
			TimerStateFeedback(IN:=FALSE);
			WasInGear := FALSE;
			iSubState := 0;

			IF BufferMode <> 0 THEN
				Error := TRUE;
				ErrorID := MC_ERROR_BUFFERMODE_NOT_SUPPORTED;
			ELSE
				InGear := F_AxisIsCoupled(Slave.NcToPlc.CoupleState) ;
				istate := SEL( InGear, STATE_ORDER, STATE_RUNNING);
			END_IF
		ELSE
			Error := FALSE;	(* reset at falling edge of Execute *)
			ErrorID := 0;
			CommandAborted := FALSE;
			InGear := FALSE;
		END_IF

	STATE_ORDER :
		Slave.PlcToNc.AxisModeLReal := GearRatio; (* 2008-06-02 KSt *)

		CASE iSubState OF
			0 :	(* read maximum master velocity *)
				fbAdsRead(	NETID:= TcMcGlobal.NCNETID_TCMC,
						PORT:= TcMcGlobal.NCPORT_TCMC,
						IDXGRP:=TcMcGlobal.Axis.Parameter.IDXGRP+Master.NcToPlc.AxisId,
						IDXOFFS:= TcMcGlobal.Axis.Parameter.IDXOFFS.VELOMAXIMUM,
						LEN:= SIZEOF(v_max),
						DESTADDR:= ADR(v_max),
						READ:= TRUE,
						TMOUT:= TcMcGlobal.tADSTimeOut);
				IF NOT fbAdsRead.Busy THEN
					Error := fbAdsRead.ERR;
					ErrorID := fbAdsRead.ERRID;
					fbAdsRead(READ:=FALSE);
					IF Error THEN
						iState := STATE_INITIALIZATION;
					ELSE
						iSubState := SEL(iAcceleration=0, iSubState + 2, iSubState + 1 );
					END_IF
				END_IF;

			1 :	(* read slave default acceleration *)
				fbAdsRead(	NETID:=TcMcGlobal.NCNETID_TCMC,
						PORT:= TcMcGlobal.NCPORT_TCMC,
						IDXGRP:=TcMcGlobal.Axis.Parameter.IDXGRP+Slave.NcToPlc.AxisId,
						IDXOFFS:= TcMcGlobal.Axis.Parameter.IDXOFFS.ACC,
						LEN:= SIZEOF(iAcceleration),
						DESTADDR:= ADR(iAcceleration),
						READ:= TRUE,
						TMOUT:= TcMcGlobal.tADSTimeOut);
				IF NOT fbAdsRead.Busy THEN
					Error := fbAdsRead.ERR;
					ErrorID := fbAdsRead.ERRID;
					fbAdsRead(READ:=FALSE);
					IF Error THEN
						iState := STATE_INITIALIZATION;
					ELSE
						iSubState := iSubState + 1;
					END_IF
				END_IF;

			2 : (* couple with dynamic gear ratio *)
				(* 	pa entspricht indirekt, naemlich bezogen auf eine maximale
					Mastergeschwindigkeit, einer maximal erlaubten 
					Beschleunigung (pa = aSlaveMax / vMasterMax ). 
					Der Begrenzungsparameter pa entspricht dabei dem 
					Kehrwert der Hochlaufzeit tH = 1 / pa . 
				*)
				IF iAcceleration > 0 AND v_max > 0 THEN
					pa_limit := iAcceleration / v_max;
				ELSE
					pa_limit := 1;
				END_IF

				sCouple.nSlaveType 	:= SEL( Options.CCVmode,
					TCNC_SLAVETYPE_LINEAR_CYCLICCHANGES_RAMP,
					TCNC_SLAVETYPE_CONST_SURFACEVELO_RAMP);
				sCouple.nMasterAxisId	:= Master.NcToPlc.AxisId;
				sCouple.nMasterSubIdx	:= 0;
				sCouple.nSlaveSubIdx		:= 0;
				sCouple.fCoupleParam1	:= pa_limit;
				sCouple.fCoupleParam2	:= 0;(* unused *)
				sCouple.fCoupleParam3	:= 0;(* unused *)
				sCouple.fCoupleParam4	:= 0;(* unused *)

				(* Slave.PlcToNc.AxisModeLReal := GearRatio;*) (* 2008-06-02 KSt *)

				fbAdsWrite(	NETID:= TcMcGlobal.NCNETID_TCMC,
						PORT:= TcMcGlobal.NCPORT_TCMC_COUPLING,
						IDXGRP:=TcMcGlobal.Axis.Functions.IDXGRP+Slave.NcToPlc.AxisId,
						IDXOFFS:= TcMcGlobal.Axis.Functions.IDXOFFS.CPL,
						LEN:= SIZEOF(sCouple),
						SRCADDR:= ADR(sCouple),
						WRITE:= TRUE,
						TMOUT:= TcMcGlobal.tADSTimeOut);
				IF NOT fbAdsWrite.Busy THEN
					Error := fbAdsWrite.ERR;
					ErrorID := fbAdsWrite.ERRID;
					fbAdsWrite(WRITE:=FALSE);
					IF Error THEN
						iState := STATE_INITIALIZATION;
					ELSE
						InGear := F_AxisIsCoupled(Slave.NcToPlc.CoupleState);
						iState := STATE_RUNNING;
					END_IF
				END_IF
		END_CASE

	STATE_RUNNING:  (* cyclic change of the gear ratio until decoupled or until Execute=FALSE *)
		TimerStateFeedback(IN:=TRUE, PT:=t#50ms); (* 5.7.2006 KSt *)
		Slave.PlcToNc.AxisModeLReal := GearRatio;
		InGear := F_AxisIsCoupled(Slave.NcToPlc.CoupleState) ;
		IF InGear THEN
			WasInGear := TRUE; (* feedback seen, 5.7.2006 KSt *)
		END_IF
		IF (NOT Enable OR NOT InGear) AND (WasInGear OR TimerStateFeedback.Q) THEN (* 5.7.2006 KSt *)
			(* Slave.PlcToNc.AxisModeLReal := 0;*) (* stop when still in gear but not enabled *) (* keep latest gear ratio - 2009-02-19 KSt *)
			CommandAborted := NOT InGear;
			iState := STATE_INITIALIZATION;
		END_IF;

	ELSE  (* CASE : Unknown program state *)
		Error := TRUE;
		ErrorID := 16#FFFFFFFF;
		iState:= STATE_INITIALIZATION;
END_CASE

ADSbusy := fbAdsWrite.BUSY OR fbAdsRead.BUSY;
IF iState=STATE_INITIALIZATION THEN
	(* reset Busy immediately  when sequence ends *)
	IF Busy THEN
		LastExecutionResult.Done := InGear;
		LastExecutionResult.CommandAborted := CommandAborted;
		LastExecutionResult.Error := Error;
		LastExecutionResult.ErrorID := ErrorID;
	END_IF
	Busy := FALSE;
	Active := FALSE;
END_IF
END_FUNCTION_BLOCK

(* POU MC_GearInMultiMaster, ST *)
FUNCTION_BLOCK MC_GearInMultiMaster
(*	MC_GearInDyn couples a slave axis to a master axis
 *	using a floating point gear ratio. The gear ratio can be 
 *	dynamically modified every PLC cycle as long as the 
 *	Execute input is TRUE.
 *	The acceleration input specifies the maximum slave
 *	acceleration in case of high gear ratio changes.
 *)
VAR_IN_OUT
	Master1			:	AXIS_REF;
	Master2			:	AXIS_REF;
	Master3			:	AXIS_REF;
	Master4			:	AXIS_REF;
	Slave			:	AXIS_REF;
END_VAR
VAR_INPUT
	Enable			:	BOOL;
	GearRatio1		:	LREAL := 1.0;
	GearRatio2		:	LREAL := 1.0;
	GearRatio3		:	LREAL := 1.0;
	GearRatio4		:	LREAL := 1.0;
	Acceleration		:	LREAL;
	Deceleration		:	LREAL;	(* not used *)
	Jerk				:	LREAL;	(* not used *)
	BufferMode		:	MC_BufferMode;	(* E *)
	Options			: 	ST_GearInMultiMasterOptions;	(* V *)	(* optional parameters *)
END_VAR
VAR_OUTPUT
	InGear				:	BOOL;
	Busy				: 	BOOL;
	Active				: 	BOOL;
	CommandAborted		:	BOOL;
	Error				:	BOOL;
	ErrorID				:	UDINT;
END_VAR
VAR
	ADSbusy			: 	BOOL;
	iState				:	_E_TcMC_STATES := STATE_INITIALIZATION;
	fbAdsWrite			:	ADSWRITE;
	sCouple				:	_ST_TcNC_CoupleSlaveMultiMaster;
	iAcceleration			: 	LREAL;
	WasInGear			:	 BOOL;
	LastExecutionResult: 	_ST_FunctionBlockResults;
END_VAR
{library private}
VAR
	TimerStateFeedback	: 	TON;
END_VAR
CASE iState OF
	STATE_INITIALIZATION:	(* *)
		Busy := FALSE;
		Active := FALSE;
		IF Enable THEN
			Busy := TRUE;
			Active := TRUE;
			fbAdsWrite(WRITE:=FALSE);
			(* initialize output values *)
			iAcceleration := Acceleration;
			ErrorID := 0;
			Error := FALSE;
			LastExecutionResult.Done := FALSE;
			LastExecutionResult.CommandAborted := FALSE;
			LastExecutionResult.Error := FALSE;
			LastExecutionResult.ErrorID := 0;
			TimerStateFeedback(IN:=FALSE);
			WasInGear := FALSE;

			IF BufferMode <> 0 THEN
				Error := TRUE;
				ErrorID := MC_ERROR_BUFFERMODE_NOT_SUPPORTED;
			ELSE
				InGear := F_AxisIsCoupled(Slave.NcToPlc.CoupleState) ;
				istate := SEL( InGear, STATE_ORDER, STATE_RUNNING);
			END_IF

		ELSE
			Error := FALSE;	(* reset when Enable is FALSE *)
			ErrorID := 0;
			CommandAborted := FALSE;
			InGear := FALSE;
		END_IF

	STATE_ORDER :
			(* couple with dynamic gear ratio *)
			sCouple.nSlaveType := TCNC_SLAVETYPE_LINEAR_MULTIMASTER;
			sCouple.nMasterSubIdx	:= 0;
			sCouple.nSlaveSubIdx		:= 0;
(*			sCouple.fCoupleParam1	:= iAcceleration;*)
			sCouple.nMasterAxisId := Master1.NcToPlc.AxisId;
			sCouple.nMasterID2 := Master2.NcToPlc.AxisId;
			sCouple.nMasterID3 := Master3.NcToPlc.AxisId;
			sCouple.nMasterID4 := Master4.NcToPlc.AxisId;
			sCouple.fSlaveAcceleration := iAcceleration;
(* 			sCouple.nCheckAndOpMode := ? *)

			(* cyclic data *)
			Slave.PlcToNc.GearRatio1 := GearRatio1;
			Slave.PlcToNc.GearRatio2 := GearRatio2;
			Slave.PlcToNc.GearRatio3 := GearRatio3;
			Slave.PlcToNc.GearRatio4 := GearRatio4;

			fbAdsWrite(	NETID:= TcMcGlobal.NCNETID_TCMC,
					PORT:= TcMcGlobal.NCPORT_TCMC_COUPLING,
					IDXGRP:=TcMcGlobal.Axis.Functions.IDXGRP+Slave.NcToPlc.AxisId,
					IDXOFFS:= TcMcGlobal.Axis.Functions.IDXOFFS.CPL,
					LEN:= SIZEOF(sCouple),
					SRCADDR:= ADR(sCouple),
					WRITE:= TRUE,
					TMOUT:= TcMcGlobal.tADSTimeOut);
			IF NOT fbAdsWrite.Busy THEN
				Error := fbAdsWrite.ERR;
				ErrorID := fbAdsWrite.ERRID;
				fbAdsWrite(WRITE:=FALSE);
				IF Error THEN
					iState := STATE_INITIALIZATION;
				ELSE
					InGear := F_AxisIsCoupled(Slave.NcToPlc.CoupleState);
					iState := STATE_RUNNING;
				END_IF
			END_IF

	STATE_RUNNING:  (* cyclic change of the gear ratio until decoupled or until Execute=FALSE *)
		TimerStateFeedback(IN:=TRUE, PT:=t#50ms); (* 5.7.2006 KSt *)
		Slave.PlcToNc.GearRatio1 := GearRatio1;
		Slave.PlcToNc.GearRatio2 := GearRatio2;
		Slave.PlcToNc.GearRatio3 := GearRatio3;
		Slave.PlcToNc.GearRatio4 := GearRatio4;
		InGear := F_AxisIsCoupled(Slave.NcToPlc.CoupleState) ;
		IF InGear THEN
			WasInGear := TRUE; (* feedback seen, 5.7.2006 KSt *)
		END_IF
		IF (NOT Enable OR NOT InGear) AND (WasInGear OR TimerStateFeedback.Q) THEN (* 5.7.2006 KSt *)
(*  keep latest gear ratio - 2008-02-19 KSt *)
			(* stop when still in gear but not enabled *)
(*			Slave.PlcToNc.GearRatio1 := 0;
			Slave.PlcToNc.GearRatio2 := 0;
			Slave.PlcToNc.GearRatio3 := 0;
			Slave.PlcToNc.GearRatio4 := 0;
*)
			CommandAborted := NOT InGear;
			iState := STATE_INITIALIZATION;
		END_IF;

	ELSE  (* CASE : Unknown program state *)
		Error := TRUE;
		ErrorID := 16#FFFFFFFF;
		iState:= STATE_INITIALIZATION;
END_CASE

ADSbusy := fbAdsWrite.BUSY;
IF iState=STATE_INITIALIZATION THEN
	(* reset Busy immediately  when sequence ends *)
	IF Busy THEN
		LastExecutionResult.Done := InGear;
		LastExecutionResult.CommandAborted := CommandAborted;
		LastExecutionResult.Error := Error;
		LastExecutionResult.ErrorID := ErrorID;
	END_IF
	Busy := FALSE;
	Active := FALSE;
END_IF
END_FUNCTION_BLOCK

(* POU MC_GearOut, ST *)
FUNCTION_BLOCK MC_GearOut
(*	This Function Block disengages the Slave axis from the Master axis immediately
	Notes:
	It is assumed that this command is followed by another command, for instance 
	MC_Stop, MC_GearIn, or any other command. If there is no new command, the 
	default condition should be: maintain last velocity.
 *)
VAR_IN_OUT
	Slave			:	AXIS_REF;	(* B *)
END_VAR
VAR_INPUT
	Execute			:	BOOL;		(* B *)
	Options			: 	ST_GearOutOptions;	(* V *)	(* optional parameters *)
END_VAR
VAR_OUTPUT
	Done			:	BOOL;		(* B *)
	Busy			: 	BOOL;		(* E *)
	Error			:	BOOL;		(* B *)
	ErrorID			:	UDINT;		(* E *)
END_VAR
VAR
	LastExecutionResult: 	_ST_FunctionBlockResults;
	ADSbusy		: 	BOOL;
	iState			:	_E_TcMC_STATES := STATE_INITIALIZATION;
	fbAdsWrite		:	ADSWRITE;
END_VAR
{library private}
VAR
	fbOnTrigger		:	R_TRIG;
END_VAR
 fbOnTrigger(CLK:= Execute);

CASE iState OF
	STATE_INITIALIZATION:	(* *)
		Busy := FALSE;
		IF NOT Execute THEN
			Done := FALSE;
			Error := FALSE;			(* reset at falling edge of Execute *)
			ErrorID := 0;
		END_IF
	    	IF fbOnTrigger.Q THEN
			(* initialize output values *)
	    		Busy := TRUE;
			Done := FALSE;
			ErrorID := 0;
			Error := FALSE;
			LastExecutionResult.Done := FALSE;
			LastExecutionResult.CommandAborted := FALSE;
			LastExecutionResult.Error := FALSE;
			LastExecutionResult.ErrorID := 0;
			fbAdsWrite(WRITE := FALSE);

			fbAdsWrite(	NETID:=TcMcGlobal.NCNETID_TCMC,
						PORT:= TcMcGlobal.NCPORT_TCMC_COUPLING, (* 12.7.2006 KSt *)
						IDXGRP:=TcMcGlobal.Axis.Functions.IDXGRP+Slave.NcToPlc.AxisId,
						IDXOFFS:= TcMcGlobal.Axis.Functions.IDXOFFS.DECPL,
						LEN:= 0,
						SRCADDR:= 0,
						WRITE:= TRUE,
						TMOUT:= TcMcGlobal.tADSTimeOut);
	
			iState := STATE_ORDER;
		END_IF;

	STATE_ORDER:
		fbAdsWrite();
		IF NOT fbAdsWrite.BUSY THEN
			IF fbAdsWrite.Err THEN
				Error := TRUE;
				ErrorID := fbAdsWrite.ErrId;
				fbAdsWrite(WRITE := FALSE);
				iState := STATE_INITIALIZATION;
			ELSE
				Done := TRUE;
				fbAdsWrite(WRITE := FALSE);
				iState := STATE_INITIALIZATION;
			END_IF;
		END_IF;

	ELSE  (* CASE : Unknown program state *)
		Error := TRUE;
		ErrorID := 16#FFFFFFFF;
		iState:= STATE_INITIALIZATION;
END_CASE

ADSbusy := fbAdsWrite.BUSY;

IF iState=STATE_INITIALIZATION THEN
	(* reset Busy immediately  when sequence ends *)
	IF Busy THEN
		LastExecutionResult.Done := Done;
		LastExecutionResult.Error := Error;
		LastExecutionResult.ErrorID := ErrorID;
	END_IF
	Busy := FALSE;
END_IF
END_FUNCTION_BLOCK

(* POU MC_Halt, FBD *)
FUNCTION_BLOCK MC_Halt
(*	This function block commands a controlled motion stop. The axis is moved to
	the state 'DiscreteMotion', until the velocity is zero. With the Done output set, the 
	state is transferred to StandStill.

	Notes:
	- MC_Halt is used to stop the axis under normal operation conditions. 
	  In non-buffered mode it is possible to set another motion command during 
	  deceleration of the axis, which will abort the MC_Halt and will be executed 
	  immediately.
	- If this command is active the next command can be issued. 
	  E.g. a driverless vehicle detects an obstacle and needs to stop. 
	  MC_Halt is issued. Before the standstill is reached the obstacle is 
	  removed and the motion can be continued by setting another motion 
	  command, so the vehicle does not stop.
*)
VAR_IN_OUT
	Axis				:	AXIS_REF;	(* B *)
END_VAR
VAR_INPUT
	Execute			:	BOOL;	(* B *)
	Deceleration		:	LREAL;	(* E *)
	Jerk				:	LREAL;	(* E *)
	BufferMode		:	MC_BufferMode;	(* E *)
	Options			: 	ST_MoveOptions;	(* optional parameters *)
END_VAR
VAR_OUTPUT
	Done			:	BOOL;	(* B *)
	Busy			: 	BOOL;	(* E *)
	Active			: 	BOOL;	(* E *)
	CommandAborted	:	BOOL;	(* E *)
	Error			:	BOOL;	(* B *)
	ErrorID			:	UDINT;	(* E *)
END_VAR
VAR
	LastExecutionResult: 	_ST_FunctionBlockResults;
	ADSbusy		: 	BOOL;
	MoveGeneric		: 	_FB_MoveUniversalGeneric;
	CmdNo: UINT;
END_VAR
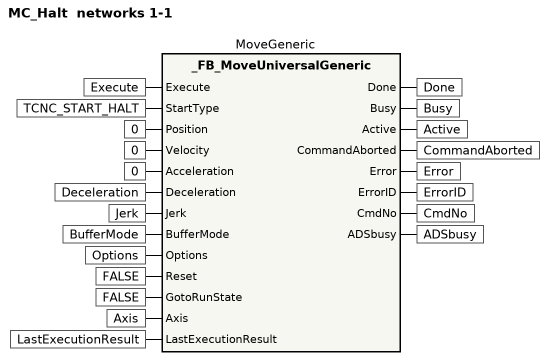
_FBD_ (* Function Block Diagram *)
NETWORK 1
	MoveGeneric   :_FB_MoveUniversalGeneric(Execute: Execute, StartType: TCNC_START_HALT, Position: 0, Velocity: 0, Acceleration: 0, Deceleration: Deceleration, Jerk: Jerk, BufferMode: BufferMode, Options: Options, Reset: FALSE, GotoRunState: FALSE, Axis: Axis, LastExecutionResult: LastExecutionResult, Busy => Busy, Active => Active, CommandAborted => CommandAborted, Error => Error, ErrorID => ErrorID, CmdNo => CmdNo, ADSbusy => ADSbusy) => Done
_END_FBD_
(* the same logic as Structured Text *)
(* Network 1 *)
MoveGeneric   (Execute := Execute, StartType := TCNC_START_HALT, Position := 0, Velocity := 0, Acceleration := 0, Deceleration := Deceleration, Jerk := Jerk, BufferMode := BufferMode, Options := Options, Reset := FALSE, GotoRunState := FALSE, Axis := Axis, LastExecutionResult := LastExecutionResult);
Busy := MoveGeneric   .Busy;
Active := MoveGeneric   .Active;
CommandAborted := MoveGeneric   .CommandAborted;
Error := MoveGeneric   .Error;
ErrorID := MoveGeneric   .ErrorID;
CmdNo := MoveGeneric   .CmdNo;
ADSbusy := MoveGeneric   .ADSbusy;
Done := MoveGeneric   .Done;
END_FUNCTION_BLOCK

(* POU MC_Home, ST *)
FUNCTION_BLOCK MC_Home
(*
	Function block defined by PLCopen Part 1 - Function blocks for motion control

	This Function Block commands the axis to perform the «search home» sequence.
	The details of this sequence can be set by the axis’ parameters. 
	The 'Position' input is used to set the absolute position when reference signal 
	is detected. This Function Bock completes at 'StandStill'.
*)
VAR_IN_OUT
	Axis				:	AXIS_REF;	(* B *)
END_VAR
VAR_INPUT
	Execute			:	BOOL;	(* B *)
	Position			:	LREAL	(* B *) := DEFAULT_HOME_POSITION;
	HomingMode		: 	MC_HomingMode;	(* E *)
	BufferMode		:	MC_BufferMode;		(* E *)
	Options			: 	ST_HomingOptions;	(* V *)	(* Beckhoff proprietary input *)
	bCalibrationCam 	: 	BOOL;	(* V *)	(* Beckhoff proprietary input *)
END_VAR
VAR_OUTPUT
	Done			:	BOOL;	(* B *)
	Busy			: 	BOOL;	(* E *)
	Active			: 	BOOL;	(* E *)
	CommandAborted	:	BOOL;	(* E *)
	Error			:	BOOL;	(* B *)
	ErrorID			:	UDINT;	(* E *)
END_VAR
VAR
	LastExecutionResult: 	_ST_FunctionBlockResults;
	ADSbusy		: 	BOOL;
	iState			: 	_E_TcMC_STATES := STATE_INITIALIZATION;
	iSubState		: 	INT;
	fbAdsWriteCmd	: 	ADSWRITE;
	fbAdsWriteRefPos: 	ADSWRITE;
	fbAdsReadRefPos: 	ADSREAD;
	ReferenceFlagValue: UDINT;
	fbSetPosition: MC_SetPosition;
	NcHomePosition 	:	LREAL;
END_VAR
{library private}
VAR
	fbTrigger			:	R_TRIG;
	fbTimeOut		:	TON;
END_VAR
 fbTrigger(CLK:= Execute);

CASE iSubState OF
	0 :	(* init *)
		iState := STATE_INITIALIZATION;	(* *)
		Busy := FALSE;
		IF NOT Execute THEN
			Done := FALSE;
			CommandAborted := FALSE;
			Error := FALSE;			(* reset at falling edge of Execute *)
			ErrorID := 0;
		END_IF
	   	IF fbTrigger.Q THEN
			(* initialize output values *)
	   		Busy := TRUE;
			Done := FALSE;
			CommandAborted := FALSE;
			Error := FALSE;
			ErrorID := 0;
			fbAdsWriteCmd(WRITE:=FALSE);
			fbAdsWriteRefPos(WRITE:=FALSE);
			fbAdsReadRefPos(READ:=FALSE);
			fbTimeOut(IN:=FALSE);
			fbSetPosition(	Execute:= FALSE, Axis:=Axis);

			IF BufferMode <> 0 THEN
		   		Busy := FALSE;
				Error := TRUE;
				ErrorID := MC_ERROR_BUFFERMODE_NOT_SUPPORTED;
			ELSE
				CASE HomingMode OF
					MC_DefaultHoming :
						IF Position < DEFAULT_HOME_POSITION THEN
							iSubState := iSubState + 1;	(* write home position before homing *)
						ELSE
							iSubState := iSubState + 2; 	(* start homing *)
						END_IF
					MC_Direct :
						ReferenceFlagValue := 1;
						IF Position < DEFAULT_HOME_POSITION THEN
							fbSetPosition.Position := Position;
							iSubState := 10;	(* set position and reference flag *)
						ELSE
							iSubState := 9; 	(* read homing position and then set position and reference flag *)
						END_IF
					MC_ForceCalibration :
						ReferenceFlagValue := 1;
						iSubState := 11; (* set reference flag *)
					MC_ResetCalibration :
						ReferenceFlagValue := 0;
						iSubState := 11; (* set reference flag *)
				ELSE (* case *)
			   		Busy := FALSE;
					Error := TRUE;
					ErrorID := MC_ERROR_CALIBRATION_ERROR; (* homing mode not supported *)
				END_CASE
			END_IF
		END_IF

	1 :	(* write homing position *)
		fbAdsWriteRefPos(	NETID:= TcMcGlobal.NCNETID_TCMC,
							PORT:= TcMcGlobal.NCPORT_TCMC,
							IDXGRP:=TcMcGlobal.Axis.Parameter.IDXGRP+Axis.NcToPlc.AxisId,
							IDXOFFS:= TcMcGlobal.Axis.Parameter.IDXOFFS.REF_POS,
							LEN:= SIZEOF(Position),
							SRCADDR:= ADR(Position),
							WRITE:= TRUE,
							TMOUT:= TcMcGlobal.tADSTimeOut);
		IF NOT fbAdsWriteRefPos.Busy THEN
			IF fbAdsWriteRefPos.Err	THEN
				Error := fbAdsWriteRefPos.ERR;
				ErrorID := fbAdsWriteRefPos.ERRID;
				iSubState := 0;
			ELSE
				NcHomePosition := Position;
				iSubState := iSubState + 1; (* start homing *)
			END_IF
		END_IF

	2 :	(* start homing *)
		fbAdsWriteCmd(	NETID:= TcMcGlobal.NCNETID_TCMC,
						PORT:= TcMcGlobal.NCPORT_TCMC,
						IDXGRP:=TcMcGlobal.Axis.Functions.IDXGRP+Axis.NcToPlc.AxisId,
						IDXOFFS:= TcMcGlobal.Axis.Functions.IDXOFFS.CALIBR,
						LEN:= 0,
						SRCADDR:= 0,
						WRITE:= TRUE,
						TMOUT:= TcMcGlobal.tADSTimeOut);
		IF NOT fbAdsWriteCmd.Busy THEN
			IF fbAdsWriteCmd.ERR THEN
				Error := fbAdsWriteCmd.ERR;
				ErrorID := fbAdsWriteCmd.ERRID;
				iSubState := 0;
			ELSE
				fbTimeOut(IN:=TRUE, PT:=TcMcGlobal.tADSTimeOut);
				IF fbTimeOut.Q THEN
					(* calibration sequence did not start *)
					Error 	:= TRUE;
					ErrorID := MC_ERROR_CALIBRATION_ERROR; (* functional/calibration error *)
					iSubState := 0;
				END_IF;
				IF F_AxisIsCalibrating(StateDWord := Axis.NcToPlc.StateDWord) THEN
					(* calibration sequence started *)
					iState := STATE_RUNNING;
					iSubState := iSubState + 1; (* wait homing *)
				END_IF
			END_IF
		END_IF

	3 :	(* homing Busy *)
		(* wait for done in cyclic interface *)
		IF NOT F_AxisIsCalibrating(StateDWord := Axis.NcToPlc.StateDWord) THEN
			IF F_AxisIsCalibrated(StateDWord := Axis.NcToPlc.StateDWord) THEN
				Done 	:= TRUE;
			ELSE
				Error 	:= TRUE;
				ErrorID := MC_ERROR_CALIBRATION_ERROR; (* functional/calibration error *)
			END_IF;
			iSubState := 0;
		END_IF;
		IF F_AxisInErrorState(StateDWord := Axis.NcToPlc.StateDWord) THEN
			Done := FALSE;
			Error := TRUE;
			ErrorID := Axis.NcToPlc.ErrorCode; (* runtime errorcode *)
			iSubState := 0;
		END_IF;

	9 :	(* read homing position - 2009-04-17 KSt added *)
		fbAdsReadRefPos(	NETID:= TcMcGlobal.NCNETID_TCMC,
							PORT:= TcMcGlobal.NCPORT_TCMC,
							IDXGRP:=TcMcGlobal.Axis.Parameter.IDXGRP+Axis.NcToPlc.AxisId,
							IDXOFFS:= TcMcGlobal.Axis.Parameter.IDXOFFS.REF_POS,
							LEN:= SIZEOF(NcHomePosition),
							DESTADDR:= ADR(NcHomePosition),
							READ:= TRUE,
							TMOUT:= TcMcGlobal.tADSTimeOut);
		IF NOT fbAdsReadRefPos.Busy THEN
			IF fbAdsReadRefPos.Err	THEN
				Error := fbAdsReadRefPos.ERR;
				ErrorID := fbAdsReadRefPos.ERRID;
				iSubState := 0;
			ELSE
				fbSetPosition.Position := NcHomePosition;
				iSubState := iSubState + 1; (* set actual position *)
			END_IF
		END_IF

	10 :	(* Static Homing forcing position from user reference *)
		fbSetPosition.Options.ClearPositionLag:= Options.ClearPositionLag;	(* 2009-04-17 KSt - changed from TRUE to option flag*)
		fbSetPosition(
			Execute:= TRUE,
			(* Position:= Position, 2009-04-17 KSt - must be set before *)
			Mode:= FALSE,	(* absolute mode *)
			Axis:= Axis );
		IF fbSetPosition.Done THEN
			iSubState := iSubState + 1;	(* set reference flag *)
		ELSIF NOT fbSetPosition.Busy THEN
			Error := TRUE;
			ErrorID := fbSetPosition.ErrorID;
			iSubState := 0;
		END_IF

	11 : 	(* Absolute homing - Set reference flag *)
		fbAdsWriteCmd(	NETID:= TcMcGlobal.NCNETID_TCMC,
						PORT:= AMSPORT_R0_NCSAF,
						IDXGRP:= TcMcGlobal.Axis.Functions.IDXGRP+Axis.NcToPlc.AxisId,
						IDXOFFS:= TcMcGlobal.Axis.Functions.IDXOFFS.SETCALFLAG,
						LEN:= SIZEOF(ReferenceFlagValue),
						SRCADDR:= ADR(ReferenceFlagValue),
						WRITE:= TRUE,
						TMOUT:= TcMcGlobal.tADSTimeOut );
		IF NOT fbAdsWriteCmd.Busy THEN
			Error := fbAdsWriteCmd.ERR;
			ErrorID := fbAdsWriteCmd.ERRID;
			Done := NOT Error;
			iSubState := 0;
		END_IF

	ELSE (* CASE : Unknown program state *)
		Error := TRUE;
		ErrorID := 16#FFFFFFFF;
		iSubState := 0;
END_CASE

ADSbusy := fbAdsWriteCmd.BUSY OR fbAdsWriteRefPos.BUSY;

IF iSubState=0 THEN
	(* reset Busy immediately  when sequence ends *)
	IF Busy THEN
		LastExecutionResult.Done := Done;
		LastExecutionResult.CommandAborted := CommandAborted;
		LastExecutionResult.Error := Error;
		LastExecutionResult.ErrorID := ErrorID;
	END_IF
	Busy := FALSE;
ELSE
	(* copy calibration cam to interface *)
	Axis.PlcToNc.ControlDWord.5 := bCalibrationCam;
END_IF

Active := Busy;
END_FUNCTION_BLOCK

(* POU MC_SetPosition, ST *)
FUNCTION_BLOCK MC_SetPosition
(*
	Function block defined by PLCopen Part 2 - Extensions

	This Function Block shifts the coordinate system of an axis by manipulating both 
	the set-point position as well as the actual position of an axis with the same value 
	without any movement caused. (Re-calibration with same following error). 
	This can be used for instance for a reference situation. This Function Block can 
	be used during motion without changing the commanded position, which is now 
	positioned in the shifted coordinate system.
*)
VAR_IN_OUT
	Axis			:	AXIS_REF;	(* B *)	(* Identifies the axis to work upon *)
END_VAR
VAR_INPUT
	Execute		:	BOOL;		(* B *)	(* Start setting position in axis *)
	Position		:	LREAL;		(* B *)	(* Position unit [u] (Means ‘Distance’ if Mode = RELATIVE) *)
	Mode		: 	BOOL;		(* E *)	(* RELATIVE =True, ABSOLUTE = False (Default) *)
	Options		:	ST_SetPositionOptions;	(* V *)	(* Beckhoff proprietary input *)
END_VAR
VAR_OUTPUT
	Done		:	BOOL;		(* B *)	(* Position has new value *)
	Busy		:	BOOL;		(* E *)	(* Shows that the Function Block is not finished *)
	Error		:	BOOL;		(* B *)	(* Signals that an error has occurred within the Function Block *)
	ErrorID		:	UDINT;		(* E *)	(* Error identification *)
END_VAR
(*
	Note:
	RELATIVE means that Position is added to the actual position value of the axis 
	at the time of execution. This results in a recalibration by a specified distance. 
	ABSOLUTE means that the actual position value of the axis is set to the value 
	specified in the Position parameter.
	When changing the position on the fly, RELATIVE mode is supposed to be preferred
*)
VAR
	ADSbusy	: 	BOOL;
	stSetPos		:	_ST_TcNC_SetPosOnTheFly;
	iState		:	_E_TcMC_STATES := STATE_INITIALIZATION;
	fbAdsWrite	:	ADSWRITE;
END_VAR
{library private}
VAR
	fbOnTrigger	:	R_TRIG;
END_VAR
fbOnTrigger(CLK:= Execute);

CASE iState OF
STATE_INITIALIZATION:
	Busy := FALSE;
	IF NOT Execute THEN
		Done := FALSE;
		Error := FALSE;			(* reset at falling edge of Execute *)
		ErrorID := 0;
	END_IF
	IF fbOnTrigger.Q THEN
		Busy := TRUE;
		(* initialize output values *)
		Done := FALSE;
		Error := FALSE;
		ErrorID := 0;
		fbAdsWrite(WRITE := FALSE);

		(* fill structure*)
		stSetPos.fNewActualPos := Position;
		stSetPos.nCtrlDWord.0 := SEL( Options.ClearPositionLag, FALSE, TRUE ); 		(* set bit 0 to clear the lag *)
		stSetPos.nCtrlDWord.1 := SEL( Options.SelectEncoderIndex, FALSE, TRUE ); 	(* set bit 1 to explicitly select an encoder / control loop - KSt 2009-04-09 *)
		stSetPos.nReserved[1]:=0;
		stSetPos.nReserved[2]:=0;

		IF Mode THEN
			(* relative mode *)
			stSetPos.nPosSetType := TCNC_POSSETTYPE_RELATIVE;
			stSetPos.fPreviousActualPos := 0;	(* value not used any longer since 2009-01-28 *)
		ELSE
			(* absolute mode *)
			stSetPos.nPosSetType := TCNC_POSSETTYPE_ABSOLUTE;
			stSetPos.fPreviousActualPos := Axis.NcToPlc.ActPos;	(* value not used any longer since 2009-01-28 *)
		END_IF

		IF Options.SelectEncoderIndex THEN (* KSt 2009-04-09 *)
			(* select the user defined encoder/control loop explicitly *)
			fbAdsWrite.IDXOFFS:= TcMcGlobal.Axis.Functions.IDXOFFS.SETPOSONTHEFLY + Options.EncoderIndex * 16#00100000;
		ELSE
			(* select the encoder / control loop that is defined by the AXIS_REF interface
				0  	=  select active encoder / control loop		- used when standard AXIS_REF interface is used
				1..n 	=  explicit encoder / control loop selection 	- used when dedicated encoder AXIS_REF interface is used 		*)
			fbAdsWrite.IDXOFFS:= TcMcGlobal.Axis.Functions.IDXOFFS.SETPOSONTHEFLY + Axis.NcToPlc.ControlLoopIndex * 16#00100000;
		END_IF

		fbAdsWrite(	NETID:= TcMcGlobal.NCNETID_TCMC,
					PORT:= AMSPORT_R0_NCSAF,
					IDXGRP:=TcMcGlobal.Axis.Functions.IDXGRP + Axis.NcToPlc.AxisId,
(*					IDXOFFS:= TcMcGlobal.Axis.Functions.IDXOFFS.SETPOSONTHEFLY + Options.EncoderIndex * 16#100000, *)(* add sub index - KSt 2008-10-22 *)
(*					IDXOFFS:= TcMcGlobal.Axis.Functions.IDXOFFS.SETPOSONTHEFLY, *)	(* see selection above - KSt 2009-04-09 *)
					LEN:= SIZEOF(stSetPos),
					SRCADDR:= ADR(stSetPos),
					WRITE:= TRUE,
					TMOUT:= TcMcGlobal.tADSTimeOut);
		iState := STATE_ORDER;
	END_IF;

STATE_ORDER:
	fbAdsWrite();
	IF NOT fbAdsWrite.Busy THEN
		IF fbAdsWrite.Err THEN
			ErrorID := fbAdsWrite.ErrId;
			Error := TRUE;
		ELSE
			Done := TRUE;
		END_IF;
		fbAdsWrite(WRITE := FALSE);
		iState := STATE_INITIALIZATION;
	END_IF;

ELSE  (* CASE : Unknown program state *)
	Error := TRUE;
	ErrorID := 16#FFFFFFFF;
	iState:= STATE_INITIALIZATION;
END_CASE

ADSbusy := fbAdsWrite.BUSY;

IF iState=STATE_INITIALIZATION THEN
	(* reset Busy immediately  when sequence ends *)
	Busy := FALSE;
END_IF
END_FUNCTION_BLOCK

(* POU MC_Jog, ST *)
FUNCTION_BLOCK MC_Jog
(*	This function block commands a jogged movement to an axis.*)
VAR_IN_OUT
	Axis				:	AXIS_REF;
END_VAR
VAR_INPUT
	JogForward 		: 	BOOL;
	JogBackwards 	: 	BOOL;
	Mode			: 	E_JogMode;
	Position 			: 	LREAL;
	Velocity			:	LREAL;
	Acceleration		:	LREAL;
	Deceleration		:	LREAL;
	Jerk				:	LREAL;
(*	BufferMode		:	MC_BufferMode;*)(* E *)
END_VAR
VAR_OUTPUT
	Done			:	BOOL;
	Busy 			:	BOOL;
	Active 			:	BOOL;
	CommandAborted	:	BOOL;
	Error			:	BOOL;
	ErrorID			:	UDINT;
END_VAR
VAR
	state: INT;
	LastExecutionResult: _ST_FunctionBlockResults;
	StateDWord: BOOL;
END_VAR
{library private}
VAR
	ExecuteMoveVelocity: BOOL;
	MoveVelocity: MC_MoveVelocity;
	MoveVelocityOut : ST_McOutputs;
	Direction: MC_Direction;

	ExecuteHalt: BOOL;
	Halt: MC_Halt;
	HaltOut : ST_McOutputs;

	ExecuteMoveAbsolute: BOOL;
	MoveAbsolute: MC_MoveAbsolute;
	MoveAbsoluteOut : ST_McOutputs;

	ExecuteMoveRelative: BOOL;
	MoveRelative : MC_MoveRelative;
	MoveRelativeOut : ST_McOutputs;

	JogMove: _FB_MoveUniversalGeneric;
	LastJogMoveResult: _ST_FunctionBlockResults;
	ExecuteJogMove: BOOL;
	StartType: _E_TCNC_StartPosType;
	JogMoveOut : ST_McOutputs;

	JogEnd: BOOL;
	TargetPosition: LREAL;
	modulo: LREAL;
END_VAR
ActCheckJogEnd;

CASE state OF
	0 : (* Initialization *)
		Busy := FALSE;
		Active := FALSE;
		ExecuteMoveVelocity := FALSE;
		ExecuteMoveRelative := FALSE;
		ExecuteMoveAbsolute := FALSE;
		ExecuteJogMove := FALSE;
		ExecuteHalt := FALSE;

		IF NOT JogForward AND NOT JogBackwards THEN (* 2009-03-12 *)
			Done := FALSE;
			CommandAborted := FALSE;
			Error := FALSE;
			ErrorID := 0;
		ELSIF (JogForward OR JogBackwards) AND F_AxisInProtectedMode(Axis.NcToPlc.StateDWord) THEN(* 2009-11-18 KSt *)
			(* MC_Jog cannot be used in protected mode (e. g. slave axis) *)
			Error := TRUE;
			ErrorID := MC_ERROR_AXIS_IN_PROTECTED_MODE;
		ELSIF JogForward AND NOT JogBackwards THEN
			Done := FALSE;
			Busy := TRUE;
			CommandAborted := FALSE;
			Error := FALSE;
			ErrorID := 0;
			Direction := MC_Positive_Direction;
			CASE Mode OF
				MC_JOGMODE_STANDARD_SLOW :
					StartType := TCNC_START_ENDLESSPLUS_SLOWMANUAL;
					ExecuteJogMove := TRUE;
					state := 3;
				MC_JOGMODE_STANDARD_FAST :
					StartType := TCNC_START_ENDLESSPLUS_FASTMANUAL;
					ExecuteJogMove := TRUE;
					state := 3;
				MC_JOGMODE_CONTINOUS :
					ExecuteMoveVelocity := TRUE;
					state := 1;
				MC_JOGMODE_INCHING :
					TargetPosition := Position;
					ExecuteMoveRelative := TRUE;
					state := 4;
				MC_JOGMODE_INCHING_MODULO :
					TargetPosition := Axis.NcToPlc.SetPos - Axis.NcToPlc.ModuloSetPos + Position;
					ExecuteMoveAbsolute := TRUE;
					state := 2;
			ELSE
				Busy := FALSE;
			END_CASE
		ELSIF JogBackwards AND NOT JogForward THEN
			Done := FALSE;
			Busy := TRUE;
			CommandAborted := FALSE;
			Error := FALSE;
			ErrorID := 0;
			Direction := MC_Negative_Direction;
			CASE Mode OF
				MC_JOGMODE_STANDARD_SLOW :
					StartType := TCNC_START_ENDLESSMINUS_SLOWMANUAL;
					ExecuteJogMove := TRUE;
					state := 3;
				MC_JOGMODE_STANDARD_FAST :
					StartType := TCNC_START_ENDLESSMINUS_FASTMANUAL;
					ExecuteJogMove := TRUE;
					state := 3;
				MC_JOGMODE_CONTINOUS :
					ExecuteMoveVelocity := TRUE;
					state := 1;
				MC_JOGMODE_INCHING :
					TargetPosition := - Position;
					ExecuteMoveRelative := TRUE;
					state := 4;
				MC_JOGMODE_INCHING_MODULO :
					modulo := Axis.NcToPlc.ModuloSetPos;
					IF modulo = 0 THEN
						TargetPosition := Axis.NcToPlc.SetPos - Position;
					ELSE
						TargetPosition := Axis.NcToPlc.SetPos - Axis.NcToPlc.ModuloSetPos;
					END_IF
					ExecuteMoveAbsolute := TRUE;
					state := 2;
			ELSE
				Busy := FALSE;
			END_CASE
		END_IF

	1 : (* continous jogging with MoveVelocity *)
		IF JogEnd THEN
			ExecuteMoveVelocity := FALSE;
			ExecuteHalt := TRUE;
		END_IF
		IF NOT MoveVelocity.Busy AND NOT Halt.Busy AND NOT F_AxisHasJob(Axis.NcToPlc.StateDWord) THEN
			Error := MoveVelocity.Error OR Halt.Error OR F_AxisInErrorState(Axis.NcToPlc.StateDWord);
			ErrorID := SEL( F_AxisInErrorState(Axis.NcToPlc.StateDWord), SEL(MoveVelocity.Error, Halt.ErrorID, MoveVelocity.ErrorID ), Axis.NcToPlc.ErrorCode);
			CommandAborted := NOT Error AND MoveVelocity.CommandAborted AND NOT ExecuteHalt; (* logic fixed 14.3.07 KSt *)
			Done := NOT Error AND NOT CommandAborted;
			ExecuteMoveVelocity := FALSE;
			ExecuteHalt := FALSE;
			IF JogEnd OR Done THEN
				state := 0;
			ELSE
				state := 9;
			END_IF
		END_IF

	2 : (* inching with MoveAbsolute *)
		IF 	Done OR
			(NOT MoveAbsolute.Busy AND NOT F_AxisHasJob(Axis.NcToPlc.StateDWord)) THEN
			Error := MoveAbsolute.Error;
			ErrorID := MoveAbsolute.ErrorID;
			CommandAborted := MoveAbsolute.CommandAborted;
			Done := NOT Error AND NOT CommandAborted;
			ExecuteMoveAbsolute := FALSE;
			IF JogEnd THEN
				state := 0;
			ELSE
				state := 9;
			END_IF
		END_IF

	3 : (* continous jogging with system parameters *)
		IF JogEnd THEN
			ExecuteJogMove := FALSE;
			ExecuteHalt := TRUE;
		END_IF
		IF NOT JogMove.Busy AND NOT Halt.Busy AND NOT F_AxisHasJob(Axis.NcToPlc.StateDWord) THEN
			Error := JogMove.Error OR Halt.Error OR F_AxisInErrorState(Axis.NcToPlc.StateDWord);
			ErrorID := SEL( F_AxisInErrorState(Axis.NcToPlc.StateDWord), SEL(JogMove.Error, Halt.ErrorID, JogMove.ErrorID ), Axis.NcToPlc.ErrorCode);
			CommandAborted := NOT Error AND JogMove.CommandAborted AND NOT ExecuteHalt; (* logic fixed 14.3.07 KSt *)
			Done := NOT Error AND NOT CommandAborted;
			ExecuteJogMove := FALSE;
			ExecuteHalt := FALSE;
			IF JogEnd OR Done THEN
				state := 0;
			ELSE
				state := 9;
			END_IF
		END_IF

	4 : (* inching with MoveRelative *)
		IF 	Done OR
			(NOT MoveRelative.Busy AND NOT F_AxisHasJob(Axis.NcToPlc.StateDWord)) THEN
			Error := MoveRelative.Error;
			ErrorID := MoveRelative.ErrorID;
			CommandAborted := MoveRelative.CommandAborted;
			Done := NOT Error AND NOT CommandAborted;
			ExecuteMoveRelative := FALSE;
			IF JogEnd THEN
				state := 0;
			ELSE
				state := 9;
			END_IF
		END_IF

	9 :	(* wait for falling edge on execute *)
		IF JogEnd THEN
			state := 0;
		END_IF
END_CASE

ActJogMove;

IF state = 0 OR state = 9 THEN
	IF Busy THEN
		LastExecutionResult.Done := Done;
		LastExecutionResult.CommandAborted := CommandAborted;
		LastExecutionResult.Error := Error;
		LastExecutionResult.ErrorID := ErrorID;
	END_IF
	Busy := FALSE;
	Active := FALSE;
ELSIF F_AxisInProtectedMode(Axis.NcToPlc.StateDWord) THEN (* 2009-11-18 KSt *)
	(* if axis is coupled on the fly - force state machine back to state zero and signal an error *)
	state := 0;
	Error := TRUE;
	ErrorID := MC_ERROR_AXIS_IN_PROTECTED_MODE;
END_IF
END_FUNCTION_BLOCK
ACTION ActCheckJogEnd:
JogEnd := 	(NOT JogForward AND NOT JogBackwards) OR
			(NOT JogForward AND Direction=MC_Positive_Direction) OR
			(NOT JogBackwards AND Direction=MC_Negative_Direction);
END_ACTION
ACTION ActJogMove:
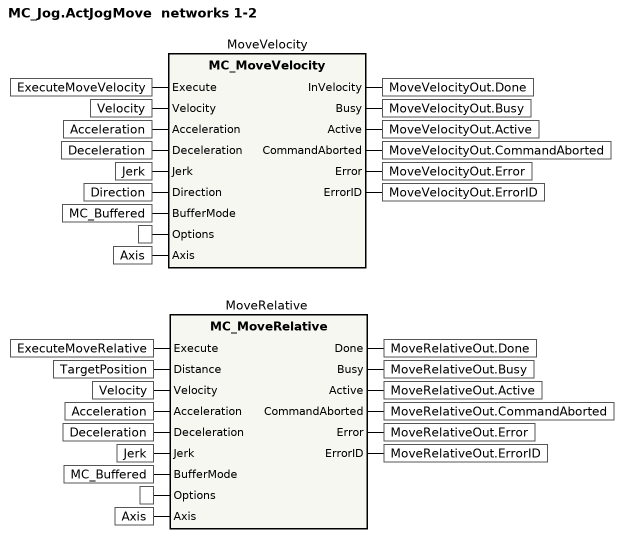
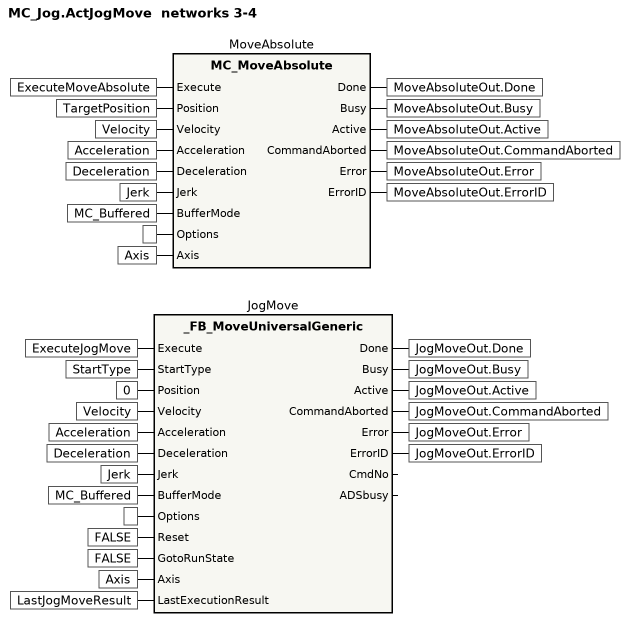
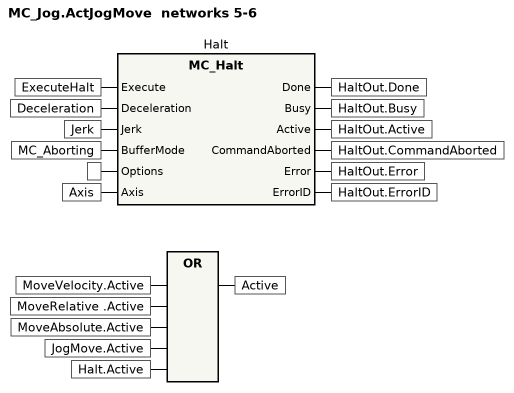
_FBD_ (* Function Block Diagram *)
NETWORK 1
	MoveVelocity:MC_MoveVelocity(Execute: ExecuteMoveVelocity, Velocity: Velocity, Acceleration: Acceleration, Deceleration: Deceleration, Jerk: Jerk, Direction: Direction, BufferMode: MC_Buffered, Options: , Axis: Axis, Busy => MoveVelocityOut.Busy, Active => MoveVelocityOut.Active, CommandAborted => MoveVelocityOut.CommandAborted, Error => MoveVelocityOut.Error, ErrorID => MoveVelocityOut.ErrorID) => MoveVelocityOut.Done
NETWORK 2
	MoveRelative :MC_MoveRelative(Execute: ExecuteMoveRelative, Distance: TargetPosition, Velocity: Velocity, Acceleration: Acceleration, Deceleration: Deceleration, Jerk: Jerk, BufferMode: MC_Buffered, Options: , Axis: Axis, Busy => MoveRelativeOut.Busy, Active => MoveRelativeOut.Active, CommandAborted => MoveRelativeOut.CommandAborted, Error => MoveRelativeOut.Error, ErrorID => MoveRelativeOut.ErrorID) => MoveRelativeOut.Done
NETWORK 3
	MoveAbsolute:MC_MoveAbsolute(Execute: ExecuteMoveAbsolute, Position: TargetPosition, Velocity: Velocity, Acceleration: Acceleration, Deceleration: Deceleration, Jerk: Jerk, BufferMode: MC_Buffered, Options: , Axis: Axis, Busy => MoveAbsoluteOut.Busy, Active => MoveAbsoluteOut.Active, CommandAborted => MoveAbsoluteOut.CommandAborted, Error => MoveAbsoluteOut.Error, ErrorID => MoveAbsoluteOut.ErrorID) => MoveAbsoluteOut.Done
NETWORK 4
	JogMove:_FB_MoveUniversalGeneric(Execute: ExecuteJogMove, StartType: StartType, Position: 0, Velocity: Velocity, Acceleration: Acceleration, Deceleration: Deceleration, Jerk: Jerk, BufferMode: MC_Buffered, Options: , Reset: FALSE, GotoRunState: FALSE, Axis: Axis, LastExecutionResult: LastJogMoveResult, Busy => JogMoveOut.Busy, Active => JogMoveOut.Active, CommandAborted => JogMoveOut.CommandAborted, Error => JogMoveOut.Error, ErrorID => JogMoveOut.ErrorID) => JogMoveOut.Done
NETWORK 5
	Halt:MC_Halt(Execute: ExecuteHalt, Deceleration: Deceleration, Jerk: Jerk, BufferMode: MC_Aborting, Options: , Axis: Axis, Busy => HaltOut.Busy, Active => HaltOut.Active, CommandAborted => HaltOut.CommandAborted, Error => HaltOut.Error, ErrorID => HaltOut.ErrorID) => HaltOut.Done
NETWORK 6
	OR(MoveVelocity.Active, MoveRelative .Active, MoveAbsolute.Active, JogMove.Active, Halt.Active) => Active
_END_FBD_
(* the same logic as Structured Text *)
(* Network 1: see the listing above *)
(* Network 2: see the listing above *)
(* Network 3: see the listing above *)
(* Network 4: see the listing above *)
(* Network 5: see the listing above *)
(* Network 6 *)
Active := MoveVelocity.Active OR (MoveRelative .Active) OR MoveAbsolute.Active OR JogMove.Active OR Halt.Active;
END_ACTION

(* POU MC_MoveVelocity, FBD *)
FUNCTION_BLOCK MC_MoveVelocity
(*	This Function Block commands a never ending controlled motion at a specified velocity. *)
VAR_IN_OUT
	Axis				:	AXIS_REF;	(* B *)
END_VAR
VAR_INPUT
	Execute			:	BOOL;	(* B *)
	Velocity			:	LREAL;	(* E *)
	Acceleration		:	LREAL;	(* E *)
	Deceleration		:	LREAL;	(* E *)
	Jerk				:	LREAL;	(* E *)
	Direction			:	MC_Direction := MC_Positive_Direction;	(* E *)
	BufferMode		:	MC_BufferMode;	(* E *)
	Options			: 	ST_MoveOptions; (* V *)
END_VAR
VAR_OUTPUT
	InVelocity		:	BOOL;	(* B *)
	Busy			: 	BOOL;	(* E *)
	Active			: 	BOOL;	(* E *)
	CommandAborted	:	BOOL;	(* E *)
	Error			:	BOOL;	(* B *)
	ErrorID			:	UDINT;	(* E *)
END_VAR
VAR
	LastExecutionResult: 	_ST_FunctionBlockResults;
	ADSbusy		: 	BOOL;
	MoveGeneric		: 	_FB_MoveUniversalGeneric;
	CmdNo: UINT;
END_VAR
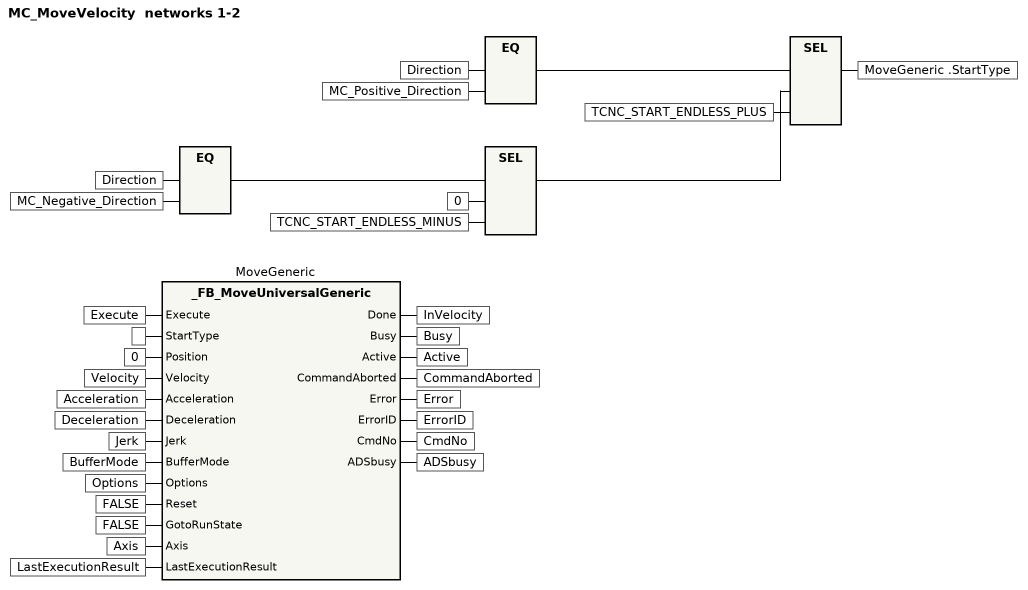
_FBD_ (* Function Block Diagram *)
NETWORK 1
	SEL(EQ(Direction, MC_Positive_Direction), SEL(EQ(Direction, MC_Negative_Direction), 0, TCNC_START_ENDLESS_MINUS), TCNC_START_ENDLESS_PLUS) => MoveGeneric .StartType
NETWORK 2
	MoveGeneric   :_FB_MoveUniversalGeneric(Execute: Execute, StartType: , Position: 0, Velocity: Velocity, Acceleration: Acceleration, Deceleration: Deceleration, Jerk: Jerk, BufferMode: BufferMode, Options: Options, Reset: FALSE, GotoRunState: FALSE, Axis: Axis, LastExecutionResult: LastExecutionResult, Busy => Busy, Active => Active, CommandAborted => CommandAborted, Error => Error, ErrorID => ErrorID, CmdNo => CmdNo, ADSbusy => ADSbusy) => InVelocity
_END_FBD_
(* the same logic as Structured Text *)
(* Network 1 *)
MoveGeneric .StartType := SEL(Direction = MC_Positive_Direction, SEL(Direction = MC_Negative_Direction, 0, TCNC_START_ENDLESS_MINUS), TCNC_START_ENDLESS_PLUS);
(* Network 2: see the listing above *)
END_FUNCTION_BLOCK

(* POU MC_MoveRelative, FBD *)
FUNCTION_BLOCK MC_MoveRelative
(*	This Function Block commands a controlled motion of a specified distance
	relative to the actual position at the time of the execution.
*)
VAR_IN_OUT
	Axis				:	AXIS_REF;	(* B *)
END_VAR
VAR_INPUT
	Execute			:	BOOL;	(* B *)
	Distance			:	LREAL;	(* B *)
	Velocity			:	LREAL;	(* E *)
	Acceleration		:	LREAL;	(* E *)
	Deceleration		:	LREAL;	(* E *)
	Jerk				:	LREAL;	(* E *)
	BufferMode		:	MC_BufferMode;	(* E *)
	Options			: 	ST_MoveOptions;	(* V *)
END_VAR
VAR_OUTPUT
	Done			:	BOOL;	(* B *)
	Busy			: 	BOOL;	(* E *)
	Active			: 	BOOL;	(* E *)
	CommandAborted	:	BOOL;	(* E *)
	Error			:	BOOL;	(* B *)
	ErrorID			:	UDINT;	(* E *)
END_VAR
VAR
	LastExecutionResult: 	_ST_FunctionBlockResults;
	ADSbusy		: 	BOOL;
	MoveGeneric		: 	_FB_MoveUniversalGeneric;
	CmdNo: UINT;
END_VAR
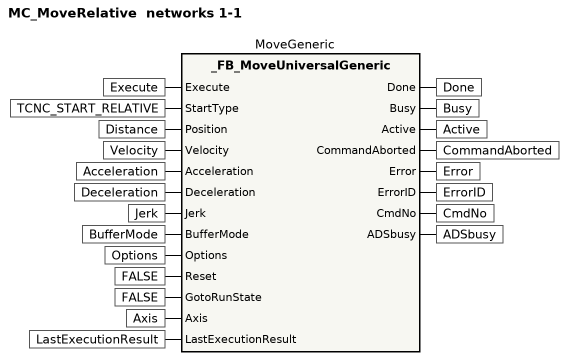
_FBD_ (* Function Block Diagram *)
NETWORK 1
	MoveGeneric   :_FB_MoveUniversalGeneric(Execute: Execute, StartType: TCNC_START_RELATIVE, Position: Distance, Velocity: Velocity, Acceleration: Acceleration, Deceleration: Deceleration, Jerk: Jerk, BufferMode: BufferMode, Options: Options, Reset: FALSE, GotoRunState: FALSE, Axis: Axis, LastExecutionResult: LastExecutionResult, Busy => Busy, Active => Active, CommandAborted => CommandAborted, Error => Error, ErrorID => ErrorID, CmdNo => CmdNo, ADSbusy => ADSbusy) => Done
_END_FBD_
(* the same logic as Structured Text *)
(* Network 1 *)
MoveGeneric   (Execute := Execute, StartType := TCNC_START_RELATIVE, Position := Distance, Velocity := Velocity, Acceleration := Acceleration, Deceleration := Deceleration, Jerk := Jerk, BufferMode := BufferMode, Options := Options, Reset := FALSE, GotoRunState := FALSE, Axis := Axis, LastExecutionResult := LastExecutionResult);
Busy := MoveGeneric   .Busy;
Active := MoveGeneric   .Active;
CommandAborted := MoveGeneric   .CommandAborted;
Error := MoveGeneric   .Error;
ErrorID := MoveGeneric   .ErrorID;
CmdNo := MoveGeneric   .CmdNo;
ADSbusy := MoveGeneric   .ADSbusy;
Done := MoveGeneric   .Done;
END_FUNCTION_BLOCK

(* POU MC_MoveAdditive, FBD *)
FUNCTION_BLOCK MC_MoveAdditive
(*	This Function Block commands a controlled motion of a specified relative
	distance additional to the most recent commanded position in the discrete 
	motion state. The most recent commanded position may be the result of a 
	previous MC_MoveAdditive motion which was aborted. If the FB is activated 
	in the Continuous Mode the specified relative distance is added to the actual 
	position at the time of the execution.

 	MC_MoveAdditive ist ähnlich MC_MoveRelative. Wenn während der Bewegung
	getriggert, dann wird allerdings die ursprüngliche Zielposition um Distance 
	verlängert. Eine Endlosachse wird in eine diskrete Bewegung ausgehend 
	von der aktuellen Position plus Distanz gewandelt.
*)
VAR_IN_OUT
	Axis				:	AXIS_REF; (* B *)
END_VAR
VAR_INPUT
	Execute			:	BOOL;	(* B *)
	Distance			:	LREAL;	(* B *)
	Velocity			:	LREAL;	(* E *)
	Acceleration		:	LREAL;	(* E *)
	Deceleration		:	LREAL;	(* E *)
	Jerk				:	LREAL;	(* E *)
	BufferMode		:	MC_BufferMode;	(* E *)
	Options			: 	ST_MoveOptions;	(* V *)
END_VAR
VAR_OUTPUT
	Done			:	BOOL;	(* B *)
	Busy			: 	BOOL;	(* E *)
	Active			: 	BOOL;	(* E *)
	CommandAborted	:	BOOL;	(* E *)
	Error			:	BOOL;	(* B *)
	ErrorID			:	UDINT;	(* E *)
END_VAR
VAR
	LastExecutionResult: 	_ST_FunctionBlockResults;
	ADSbusy		: 	BOOL;
	MoveGeneric		: 	_FB_MoveUniversalGeneric;
	CmdNo: UINT;
END_VAR
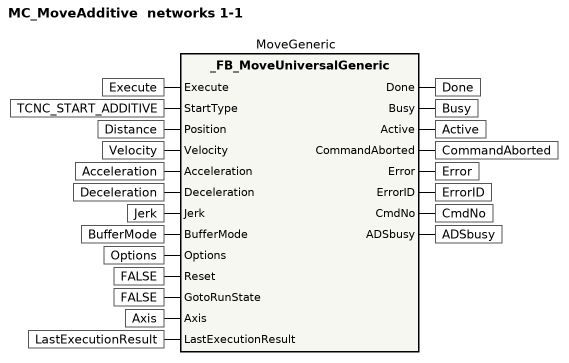
_FBD_ (* Function Block Diagram *)
NETWORK 1
	MoveGeneric  :_FB_MoveUniversalGeneric(Execute: Execute, StartType: TCNC_START_ADDITIVE, Position: Distance, Velocity: Velocity, Acceleration: Acceleration, Deceleration: Deceleration, Jerk: Jerk, BufferMode: BufferMode, Options: Options, Reset: FALSE, GotoRunState: FALSE, Axis: Axis, LastExecutionResult: LastExecutionResult, Busy => Busy, Active => Active, CommandAborted => CommandAborted, Error => Error, ErrorID => ErrorID, CmdNo => CmdNo, ADSbusy => ADSbusy) => Done
_END_FBD_
(* the same logic as Structured Text *)
(* Network 1 *)
MoveGeneric  (Execute := Execute, StartType := TCNC_START_ADDITIVE, Position := Distance, Velocity := Velocity, Acceleration := Acceleration, Deceleration := Deceleration, Jerk := Jerk, BufferMode := BufferMode, Options := Options, Reset := FALSE, GotoRunState := FALSE, Axis := Axis, LastExecutionResult := LastExecutionResult);
Busy := MoveGeneric  .Busy;
Active := MoveGeneric  .Active;
CommandAborted := MoveGeneric  .CommandAborted;
Error := MoveGeneric  .Error;
ErrorID := MoveGeneric  .ErrorID;
CmdNo := MoveGeneric  .CmdNo;
ADSbusy := MoveGeneric  .ADSbusy;
Done := MoveGeneric  .Done;
END_FUNCTION_BLOCK

(* POU MC_MoveContinuousAbsolute, FBD *)
FUNCTION_BLOCK MC_MoveContinuousAbsolute
(*	This function block commands a controlled motion to a specified absolute position
	ending with the specified velocity.

	Notes:
	- If the target is reached and no new motion command is put into the buffer, the 
	  axis continues to run with the specified ‘EndVelocity’.
	- This Function Block places the axis into the 'Continuous Motion' state, even 
	  during the initial motion by a relative distance, and remains in the 'Continuous 
	  Motion' state once the EndVelocity has been reached.

	MoveContinous ist ähnlich MoveVelocity. Es wird aber zunächst mit einem PTP-Profil
	eine Zwischenposition angefahren (mit Velocity). Ab dieser Position geht die Bewegung
	in eine Endlosfahrt mit EndVelocity über.
*)
VAR_IN_OUT
	Axis				:	AXIS_REF; (* B *)
END_VAR
VAR_INPUT
	Execute			:	BOOL;	(* B *)
	Position			:	LREAL;	(* B *)
	Velocity			:	LREAL;	(* B *)
	EndVelocity		:	LREAL;	(* B *)
	Acceleration		:	LREAL;	(* E *)
	Deceleration		:	LREAL;	(* E *)
	Jerk				:	LREAL;	(* E *)
	BufferMode		:	MC_BufferMode;	(* E *)
	Options			: 	ST_MoveOptions;
END_VAR
VAR_OUTPUT
	InEndVelocity		:	BOOL;	(* B *)
	Busy			: 	BOOL;	(* E *)
	Active			: 	BOOL;	(* E *)
	CommandAborted :	BOOL;	(* E *)
	Error			:	BOOL;	(* B *)
	ErrorID			:	UDINT;	(* E *)
END_VAR
VAR
	LastExecutionResult: 	_ST_FunctionBlockResults;
	ADSbusy		: 	BOOL;
	MoveGeneric		: 	_FB_MoveUniversalGeneric;
	CmdNo: UINT;
END_VAR
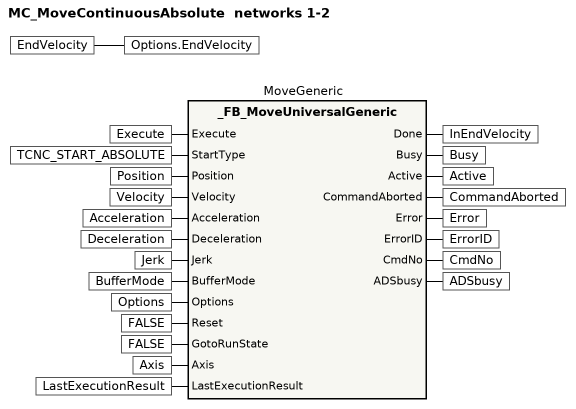
_FBD_ (* Function Block Diagram *)
NETWORK 1
	EndVelocity => Options.EndVelocity
NETWORK 2
	MoveGeneric  :_FB_MoveUniversalGeneric(Execute: Execute, StartType: TCNC_START_ABSOLUTE, Position: Position, Velocity: Velocity, Acceleration: Acceleration, Deceleration: Deceleration, Jerk: Jerk, BufferMode: BufferMode, Options: Options, Reset: FALSE, GotoRunState: FALSE, Axis: Axis, LastExecutionResult: LastExecutionResult, Busy => Busy, Active => Active, CommandAborted => CommandAborted, Error => Error, ErrorID => ErrorID, CmdNo => CmdNo, ADSbusy => ADSbusy) => InEndVelocity
_END_FBD_
(* the same logic as Structured Text *)
(* Network 1 *)
Options.EndVelocity := EndVelocity;
(* Network 2 *)
MoveGeneric  (Execute := Execute, StartType := TCNC_START_ABSOLUTE, Position := Position, Velocity := Velocity, Acceleration := Acceleration, Deceleration := Deceleration, Jerk := Jerk, BufferMode := BufferMode, Options := Options, Reset := FALSE, GotoRunState := FALSE, Axis := Axis, LastExecutionResult := LastExecutionResult);
Busy := MoveGeneric  .Busy;
Active := MoveGeneric  .Active;
CommandAborted := MoveGeneric  .CommandAborted;
Error := MoveGeneric  .Error;
ErrorID := MoveGeneric  .ErrorID;
CmdNo := MoveGeneric  .CmdNo;
ADSbusy := MoveGeneric  .ADSbusy;
InEndVelocity := MoveGeneric  .Done;
END_FUNCTION_BLOCK

(* POU MC_MoveContinuousRelative, FBD *)
FUNCTION_BLOCK MC_MoveContinuousRelative
(*	This function block commands a controlled motion of a specified relative distance
	ending with the specified velocity.

	Notes:
	- If the target is reached and no new motion command is put into the buffer, the 
	  axis continues to run with the specified ‘EndVelocity’.
	- This Function Block places the axis into the 'Continuous Motion' state, even 
	  during the initial motion by a relative distance, and remains in the 'Continuous 
	  Motion' state once the EndVelocity has been reached.

	MoveContinous ist ähnlich MoveVelocity. Es wird aber zunächst mit einem PTP-Profil
	eine Zwischenposition angefahren (mit Velocity). Ab dieser Position geht die Bewegung
	in eine Endlosfahrt mit EndVelocity über.
*)
VAR_IN_OUT
	Axis				:	AXIS_REF; (* B *)
END_VAR
VAR_INPUT
	Execute			:	BOOL;	(* B *)
	Distance			:	LREAL;	(* B *)
	Velocity			:	LREAL;	(* B *)
	EndVelocity		:	LREAL;	(* B *)
	Acceleration		:	LREAL;	(* E *)
	Deceleration		:	LREAL;	(* E *)
	Jerk				:	LREAL;	(* E *)
	BufferMode		:	MC_BufferMode;	(* E *)
	Options			: 	ST_MoveOptions;
END_VAR
VAR_OUTPUT
	InEndVelocity		:	BOOL;	(* B *)
	Busy			: 	BOOL;	(* E *)
	Active			: 	BOOL;	(* E *)
	CommandAborted :	BOOL;	(* E *)
	Error			:	BOOL;	(* B *)
	ErrorID			:	UDINT;	(* E *)
END_VAR
VAR
	LastExecutionResult: 	_ST_FunctionBlockResults;
	ADSbusy		: 	BOOL;
	MoveGeneric		: 	_FB_MoveUniversalGeneric;
	CmdNo: UINT;
END_VAR
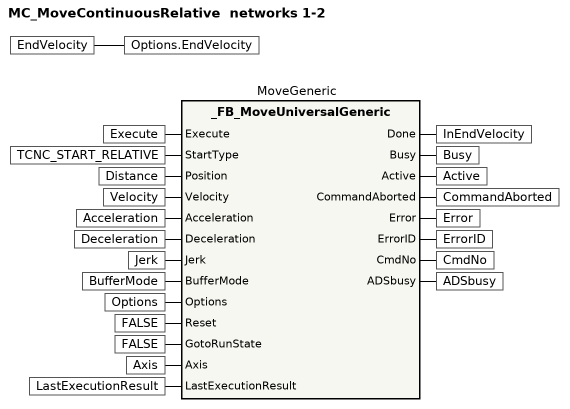
_FBD_ (* Function Block Diagram *)
NETWORK 1
	EndVelocity => Options.EndVelocity
NETWORK 2
	MoveGeneric  :_FB_MoveUniversalGeneric(Execute: Execute, StartType: TCNC_START_RELATIVE, Position: Distance, Velocity: Velocity, Acceleration: Acceleration, Deceleration: Deceleration, Jerk: Jerk, BufferMode: BufferMode, Options: Options, Reset: FALSE, GotoRunState: FALSE, Axis: Axis, LastExecutionResult: LastExecutionResult, Busy => Busy, Active => Active, CommandAborted => CommandAborted, Error => Error, ErrorID => ErrorID, CmdNo => CmdNo, ADSbusy => ADSbusy) => InEndVelocity
_END_FBD_
(* the same logic as Structured Text *)
(* Network 1 *)
Options.EndVelocity := EndVelocity;
(* Network 2 *)
MoveGeneric  (Execute := Execute, StartType := TCNC_START_RELATIVE, Position := Distance, Velocity := Velocity, Acceleration := Acceleration, Deceleration := Deceleration, Jerk := Jerk, BufferMode := BufferMode, Options := Options, Reset := FALSE, GotoRunState := FALSE, Axis := Axis, LastExecutionResult := LastExecutionResult);
Busy := MoveGeneric  .Busy;
Active := MoveGeneric  .Active;
CommandAborted := MoveGeneric  .CommandAborted;
Error := MoveGeneric  .Error;
ErrorID := MoveGeneric  .ErrorID;
CmdNo := MoveGeneric  .CmdNo;
ADSbusy := MoveGeneric  .ADSbusy;
InEndVelocity := MoveGeneric  .Done;
END_FUNCTION_BLOCK

(* POU MC_MoveModulo, ST *)
FUNCTION_BLOCK MC_MoveModulo
(* This Function Block commands a controlled motion to a specified absolute modulo position. *)
VAR_IN_OUT
	Axis				:	AXIS_REF;
END_VAR
VAR_INPUT
	Execute			:	BOOL;
	Position			:	LREAL;
	Velocity			:	LREAL;
	Acceleration		:	LREAL;
	Deceleration		:	LREAL;
	Jerk				:	LREAL;
	Direction			:	MC_Direction;	(* E *)	(* modulo shortest way, modulo positive, modulo negative *)
	BufferMode		:	MC_BufferMode;(* E *)
	Options			: 	ST_MoveOptions;
END_VAR
VAR_OUTPUT
	Done				:	BOOL;	(* B *)
	Busy				: 	BOOL;	(* E *)
	Active				: 	BOOL;	(* E *)
	CommandAborted		:	BOOL;	(* E *)
	Error				:	BOOL;	(* B *)
	ErrorID				:	UDINT;	(* E *)
END_VAR
VAR
	LastExecutionResult: _ST_FunctionBlockResults;
	ADSbusy: BOOL;
	MoveGeneric: _FB_MoveUniversalGeneric;
	StartType: UDINT;
	CmdNo: UINT;
END_VAR
CASE Direction OF
	MC_Positive_Direction:
		StartType := TCNC_START_MODULO_PLUS;
		MC_MoveModuloCall;

	MC_Shortest_Way:
		StartType := TCNC_START_MODULO_SHORT;
		MC_MoveModuloCall;

	MC_Negative_Direction:
		StartType := TCNC_START_MODULO_MINUS;
		MC_MoveModuloCall;

	MC_Current_Direction:
		StartType := TCNC_START_MODULO_CURRENT;
		MC_MoveModuloCall;
	ELSE
		IF Execute THEN
			Error := TRUE;
			ErrorID := MC_ERROR_WRONG_MODE;
		ELSE
			Error := FALSE;
			ErrorID := 0;
		END_IF
		Execute := FALSE;
		MC_MoveModuloCall;
		Done := FALSE;
		Busy := FALSE;
		Active := FALSE;
		CommandAborted := FALSE;
END_CASE
END_FUNCTION_BLOCK
ACTION MC_MoveModuloCall:
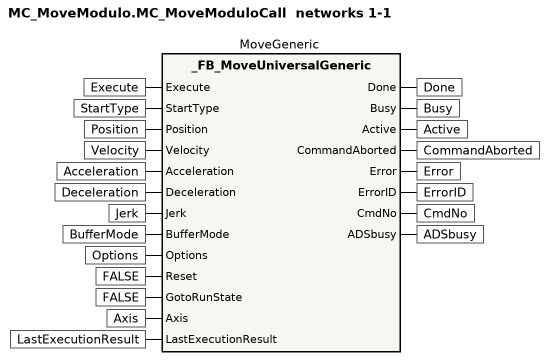
_FBD_ (* Function Block Diagram *)
NETWORK 1
	MoveGeneric :_FB_MoveUniversalGeneric(Execute: Execute, StartType: StartType, Position: Position, Velocity: Velocity, Acceleration: Acceleration, Deceleration: Deceleration, Jerk: Jerk, BufferMode: BufferMode, Options: Options, Reset: FALSE, GotoRunState: FALSE, Axis: Axis, LastExecutionResult: LastExecutionResult, Busy => Busy, Active => Active, CommandAborted => CommandAborted, Error => Error, ErrorID => ErrorID, CmdNo => CmdNo, ADSbusy => ADSbusy) => Done
_END_FBD_
(* the same logic as Structured Text *)
(* Network 1 *)
MoveGeneric (Execute := Execute, StartType := StartType, Position := Position, Velocity := Velocity, Acceleration := Acceleration, Deceleration := Deceleration, Jerk := Jerk, BufferMode := BufferMode, Options := Options, Reset := FALSE, GotoRunState := FALSE, Axis := Axis, LastExecutionResult := LastExecutionResult);
Busy := MoveGeneric .Busy;
Active := MoveGeneric .Active;
CommandAborted := MoveGeneric .CommandAborted;
Error := MoveGeneric .Error;
ErrorID := MoveGeneric .ErrorID;
CmdNo := MoveGeneric .CmdNo;
ADSbusy := MoveGeneric .ADSbusy;
Done := MoveGeneric .Done;
END_ACTION

(* POU MC_MoveSuperImposed, ST *)
(*	MC_MovedSuperimposed	(extended version 2)
 *
 *	This Function Block commands a controlled motion of a specified relative distance additional to an existing motion.
 *	The existing Motion is not interrupted, but is superimposed by the additional motion.
 *
 *	- Version 2 adds multiple modes and feedback information to the 
 *	  standard MC_MoveSuperimposed block.
 * 	- The version 2 block is compatible to the MC_MovedSuperimposed block when Mode
 *	  SUPERPOSITIONMODE_VELOREDUCTION_ADDITIVEMOTION (integer value 1) is used.
 *)
FUNCTION_BLOCK MC_MoveSuperImposed
VAR_IN_OUT
	Axis				:	AXIS_REF;	(* B *)
END_VAR
VAR_INPUT
	Execute			:	BOOL;	(* B *)
	Mode 			:	E_SuperpositionMode;	(* V *)
	Distance			:	LREAL;	(* B *)	(* distance to catch up or fall back with the superposition process *)
	VelocityDiff		:	LREAL;	(* E *)	(* maximum velocity difference - will be added or subtrated to the process velocity *)
	Acceleration		:	LREAL;	(* E *)
	Deceleration		:	LREAL;	(* E *)
	Jerk				:	LREAL;	(* E *)	(* currently not used *)
	VelocityProcess	:	LREAL;	(* V *)	(* constant velocity of the axis without superposition *)
	Length			:	LREAL;	(* V *)	(* moved distance while the superposition takes place (name has been MaxDistance before) *)
	Options			:	ST_SuperpositionOptions;	(* V *)
END_VAR
VAR_OUTPUT
	Done			:	BOOL;	(* B *)
	Busy			:	BOOL;	(* E *)
	Active			:	BOOL;	(* E *)
	CommandAborted	:	BOOL;	(* E *)
	Error			:	BOOL;	(* B *)
	ErrorID			:	UDINT;	(* E *)
	Warning			: 	BOOL;	(* V *)
	WarningId		: 	UDINT;	(* V *)
	ActualVelocityDiff	: 	LREAL;	(* V *)	(* calculated maximum velocity boost during superposition <= VelocityDiff *)
	ActualDistance	: 	LREAL;	(* V *)	(* calculated superimposed distance <= Distance*)
	ActualLength		: 	LREAL;	(* V *)	(* calculated length of the superposition <= MaxDistance *)
	ActualAcceleration : 	LREAL;	(* V *)	(* calculated acceleration during superposition *)
	ActualDeceleration : 	LREAL;	(* V *)	(* calculated deceleration during superposition *)
END_VAR
VAR
	LastExecutionResult: 	_ST_FunctionBlockResults;
	ADSbusy		: 	BOOL;
	CompensationStarted: 	BOOL;
	AxisHasJobAtStartOfCompensation	: 	BOOL; 	(* HasJob flag when starting the compensation *)
	AxisIsMovingAtStartOfCompensation	:	BOOL; 	(* Moving flag when starting the compensation *)
	iState			: 	_E_TcMC_STATES := STATE_INITIALIZATION;
	fbAdsReadWrite	: 	ADSRDWRTEX;
	sNcCompensation	:	_ST_TcNC_Compensation2;
END_VAR
{library private}
VAR
	fbTrigger			:	R_TRIG;
	fbTimeOut		: 	TON;
END_VAR
(* ====================================================================== *)
(* *)
(* ====================================================================== *)
fbTrigger(CLK:= Execute);

CASE iState OF
STATE_INITIALIZATION:	(* *)
	Busy := FALSE;
	Active := FALSE;

	IF NOT Execute THEN
		Done := FALSE;
		CommandAborted := FALSE;
		Error := FALSE;			(* reset at falling edge of Execute *)
		ErrorID := 0;
	END_IF;

    	IF fbTrigger.Q THEN
		(* initialize output values *)
		Done := FALSE;
		Busy := TRUE;
		CommandAborted := FALSE;
		Error := FALSE;
		ErrorID := 0;
		Warning := FALSE;
		WarningId := 0;
		LastExecutionResult.Done := FALSE;
		LastExecutionResult.CommandAborted := FALSE;
		LastExecutionResult.Error := FALSE;
		LastExecutionResult.ErrorID := 0;
		ActualVelocityDiff := 0;
		ActualDistance := 0;
		ActualLength := 0;
		CompensationStarted := FALSE;
		fbTimeOut(IN:= FALSE);
		fbAdsReadWrite(WRTRD:=FALSE);

		(* 2009-10-06 KSt - initial HasJob and InMotion state check *)
		AxisHasJobAtStartOfCompensation := F_AxisHasJob(Axis.NcToPlc.StateDWord);
		AxisIsMovingAtStartOfCompensation := F_AxisIsMoving(Axis.NcToPlc.StateDWord);
		(* error when ... *)
		(* 24.09.2009 HKP - Fehlerabfrage nur im Default-Fall mit  '(0) SUPERPOSITIONOPTION_ABORTATSTANDSTILL' sinnvoll *)
		(* IF  NOT F_AxisHasJob(Axis.NcToPlc.StateDWord) THEN  *) (* 12.6.2007 KSt - geändert von "NOT AxisIsMoving" nach "NOT AxisHasJob" *)
		IF  Options.AbortOption = SUPERPOSITIONOPTION_ABORTATSTANDSTILL AND NOT  F_AxisHasJob(Axis.NcToPlc.StateDWord) THEN
			ErrorID := MC_ERROR_AXIS_IS_NOT_MOVING;
			Error := TRUE;
		ELSE
			(* fill structure *)
			sNcCompensation.nCompType		:= Mode;
			sNcCompensation.fAccPlus			:= Acceleration;
			sNcCompensation.fAccMinus		:= Deceleration;
			sNcCompensation.fVeloDiff			:= VelocityDiff;
			sNcCompensation.fVeloProcess		:= VelocityProcess;
			sNcCompensation.fDistance		:= Distance;
			sNcCompensation.fLength		 	:= Length;
			(* WarningID holds optional parameters when sending the command to the NC *)
			sNcCompensation.nWarningId		:= Options.AbortOption; (* 2009-06-30 KSt *)

			fbAdsReadWrite.PORT := SEL(Axis.ADS.Port = 0, Axis.ADS.port, AMSPORT_R0_NCSAF);	(* KSt, 20090123 *)
			fbAdsReadWrite(NETID:= TcMcGlobal.NCNETID_TCMC,
							(* PORT:= TcMcGlobal.NCPORT_TCMC,*) 		(* KSt, 20090123 *)
							IDXGRP:= TcMcGlobal.Axis.Functions.IDXGRP+Axis.NcToPlc.AxisId,
							IDXOFFS:= TcMcGlobal.Axis.Functions.IDXOFFS.STARTSCOM,
							WRITELEN:= SIZEOF(sNcCompensation),
							READLEN:= SIZEOF(sNcCompensation),
							SRCADDR:= ADR(sNcCompensation),
							DESTADDR:= ADR(sNcCompensation),
							WRTRD:= TRUE,
							TMOUT:= TcMcGlobal.tADSTimeOut );

			iState := STATE_ORDER;
		END_IF;
	END_IF;

STATE_ORDER:  (* wait until command is accepted *)
	fbAdsReadWrite(WRTRD:= TRUE);
	IF NOT fbAdsReadWrite.Busy THEN
		IF fbAdsReadWrite.Err THEN
			Error := TRUE;
			ErrorID := fbAdsReadWrite.ErrId;
			iState := STATE_INITIALIZATION;
		ELSE
			IF fbAdsReadWrite.COUNT_R > 0 THEN
				ActualVelocityDiff := sNcCompensation.fVeloDiff;
				ActualDistance := sNcCompensation.fDistance;
				ActualLength := sNcCompensation.fLength;
				ActualAcceleration := sNcCompensation.fAccPlus;		(* 2010-02-25 KSt *)
				ActualDeceleration := sNcCompensation.fAccMinus;	(* 2010-02-25 KSt *)
				WarningId := sNcCompensation.nWarningId;	(* 2009-01-29 KSt *)
				Warning := WarningId <> 0;					(* 2009-01-29 KSt *)
			END_IF
			Active := TRUE;
			CompensationStarted := F_AxisIsCompensating(Axis.NcToPlc.StateDWord) ;
			iState := STATE_RUNNING;
		END_IF;
	END_IF;

STATE_RUNNING:  (* wait until axis stands still *)
	WarningId := sNcCompensation.nWarningId;
	Warning := WarningId <> 0;
(*	Busy := F_AxisIsCompensating(Axis.NcToPlc.StateDWord);
	IF Busy THEN	KSt, 29.4.2008 *)

	IF F_AxisIsCompensating(Axis.NcToPlc.StateDWord) THEN 	(* KSt, 29.4.2008 *)
		CompensationStarted := TRUE;
	ELSIF CompensationStarted  (* AND compensation finished now *) THEN
		IF AxisHasJobAtStartOfCompensation AND NOT F_AxisHasJob(Axis.NcToPlc.StateDWord) THEN (* 2009-10-06 KSt *)
			(* command aborted, move has been stopped before superposition finished because the HasJob flag turned off (KSt, 2009-08-13) *)
			CommandAborted := TRUE;
			iState := STATE_INITIALIZATION;
		ELSIF NOT AxisHasJobAtStartOfCompensation AND AxisIsMovingAtStartOfCompensation THEN (* 2009-10-06 KSt *)
			(* in case of axes coupled to actual position (encoder axes or disabled axes) *)
			IF NOT F_AxisIsMoving(Axis.NcToPlc.StateDWord) THEN (* 2009-10-06 KSt *)
				CommandAborted := TRUE;
				iState := STATE_INITIALIZATION;
			ELSE
				(* check moving state next cycle - delay is necessary since moving flag turnes off later than the compensation flag *)
				iState := STATE_WAITING;
			END_IF
		ELSE
			(* the initial HasJob or Moving state was the same as at end of compensation - assume that superposition completed *)
			Done := TRUE;
			iState := STATE_INITIALIZATION;
		END_IF
	ELSE (* compensation did not start so far *)
		(* check for superposition not beeing started (KSt, 12.01.2004) *)
		fbTimeOut(IN:= TRUE, PT:= T#50ms);
		IF fbTimeOut.Q THEN
			(*	when the ADS command comes back without any error but
				the compensation does not start anyway, we assume that  
				a very short compensation already has been executed. 
			*)
			Done := TRUE; (* after short timeout *)
			iState := STATE_INITIALIZATION;
		END_IF;
	END_IF

